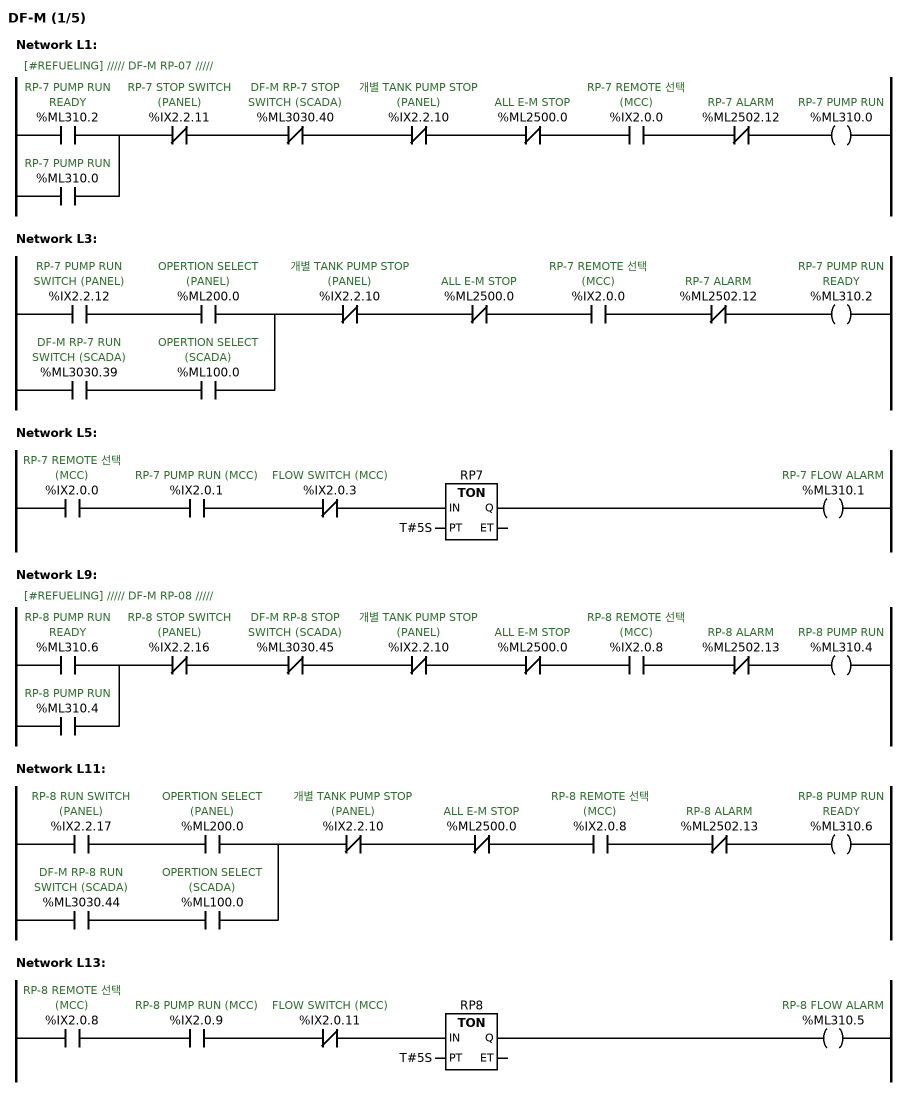
(* [#REFUELING] ///// DF-M RP-07 ///// *)
(* Rung L1 *)
%ML310.0 := (%ML310.2 OR %ML310.0) AND NOT %IX2.2.11 AND NOT %ML3030.40 AND NOT %IX2.2.10 AND NOT %ML2500.0 AND %IX2.0.0 AND NOT %ML2502.12;
(* Rung L3 *)
%ML310.2 := ((%IX2.2.12 AND %ML200.0) OR (%ML3030.39 AND %ML100.0)) AND NOT %IX2.2.10 AND NOT %ML2500.0 AND %IX2.0.0 AND NOT %ML2502.12;
(* Rung L5 *)
RP7(IN := %IX2.0.0 AND %IX2.0.1 AND NOT %IX2.0.3, PT := T#5S);
%ML310.1 := RP7.Q;
(* [#REFUELING] ///// DF-M RP-08 ///// *)
(* Rung L9 *)
%ML310.4 := (%ML310.6 OR %ML310.4) AND NOT %IX2.2.16 AND NOT %ML3030.45 AND NOT %IX2.2.10 AND NOT %ML2500.0 AND %IX2.0.8 AND NOT %ML2502.13;
(* Rung L11 *)
%ML310.6 := ((%IX2.2.17 AND %ML200.0) OR (%ML3030.44 AND %ML100.0)) AND NOT %IX2.2.10 AND NOT %ML2500.0 AND %IX2.0.8 AND NOT %ML2502.13;
(* Rung L13 *)
RP8(IN := %IX2.0.8 AND %IX2.0.9 AND NOT %IX2.0.11, PT := T#5S);
%ML310.5 := RP8.Q;

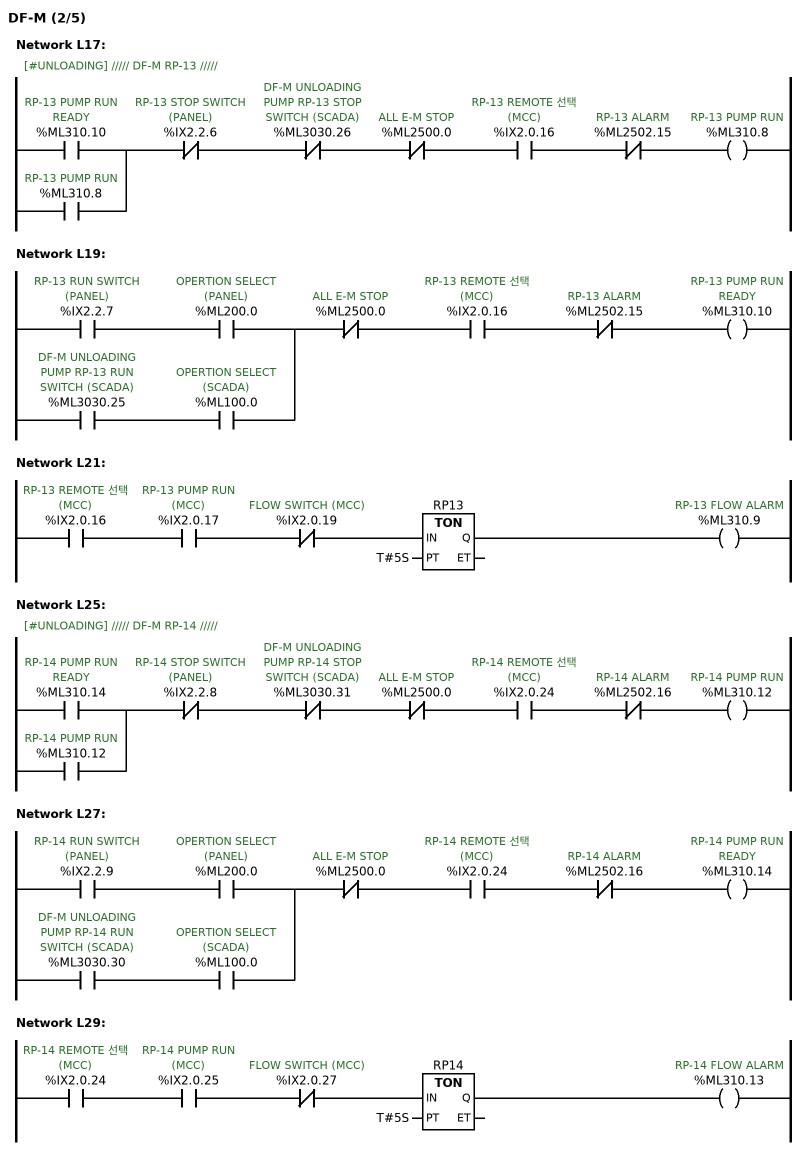
(* [#UNLOADING] ///// DF-M RP-13 ///// *)
(* Rung L17 *)
%ML310.8 := (%ML310.10 OR %ML310.8) AND NOT %IX2.2.6 AND NOT %ML3030.26 AND NOT %ML2500.0 AND %IX2.0.16 AND NOT %ML2502.15;
(* Rung L19 *)
%ML310.10 := ((%IX2.2.7 AND %ML200.0) OR (%ML3030.25 AND %ML100.0)) AND NOT %ML2500.0 AND %IX2.0.16 AND NOT %ML2502.15;
(* Rung L21 *)
RP13(IN := %IX2.0.16 AND %IX2.0.17 AND NOT %IX2.0.19, PT := T#5S);
%ML310.9 := RP13.Q;
(* [#UNLOADING] ///// DF-M RP-14 ///// *)
(* Rung L25 *)
%ML310.12 := (%ML310.14 OR %ML310.12) AND NOT %IX2.2.8 AND NOT %ML3030.31 AND NOT %ML2500.0 AND %IX2.0.24 AND NOT %ML2502.16;
(* Rung L27 *)
%ML310.14 := ((%IX2.2.9 AND %ML200.0) OR (%ML3030.30 AND %ML100.0)) AND NOT %ML2500.0 AND %IX2.0.24 AND NOT %ML2502.16;
(* Rung L29 *)
RP14(IN := %IX2.0.24 AND %IX2.0.25 AND NOT %IX2.0.27, PT := T#5S);
%ML310.13 := RP14.Q;

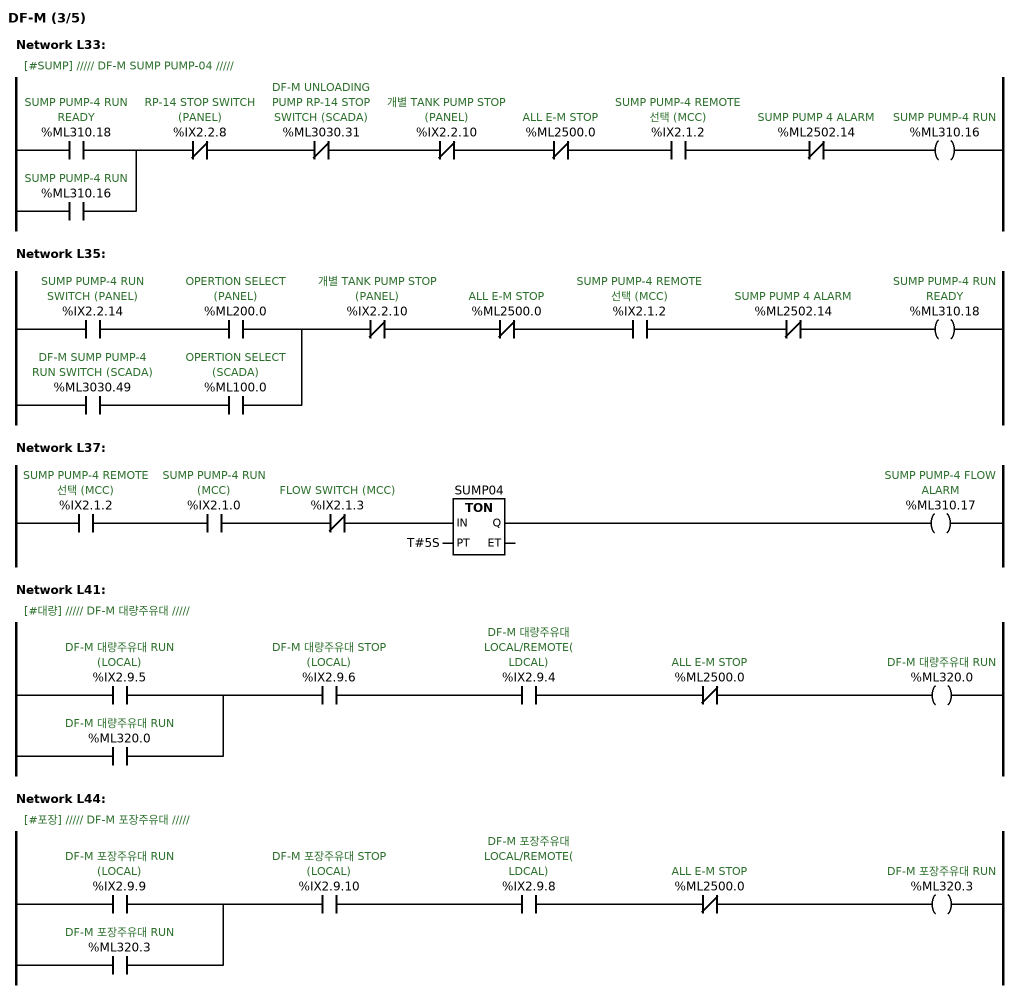
(* [#SUMP] ///// DF-M SUMP PUMP-04 ///// *)
(* Rung L33 *)
%ML310.16 := (%ML310.18 OR %ML310.16) AND NOT %IX2.2.8 AND NOT %ML3030.31 AND NOT %IX2.2.10 AND NOT %ML2500.0 AND %IX2.1.2 AND NOT %ML2502.14;
(* Rung L35 *)
%ML310.18 := ((%IX2.2.14 AND %ML200.0) OR (%ML3030.49 AND %ML100.0)) AND NOT %IX2.2.10 AND NOT %ML2500.0 AND %IX2.1.2 AND NOT %ML2502.14;
(* Rung L37 *)
SUMP04(IN := %IX2.1.2 AND %IX2.1.0 AND NOT %IX2.1.3, PT := T#5S);
%ML310.17 := SUMP04.Q;
(* [#대량] ///// DF-M 대량주유대 ///// *)
(* Rung L41 *)
%ML320.0 := (%IX2.9.5 OR %ML320.0) AND %IX2.9.6 AND %IX2.9.4 AND NOT %ML2500.0;
(* [#포장] ///// DF-M 포장주유대 ///// *)
(* Rung L44 *)
%ML320.3 := (%IX2.9.9 OR %ML320.3) AND %IX2.9.10 AND %IX2.9.8 AND NOT %ML2500.0;

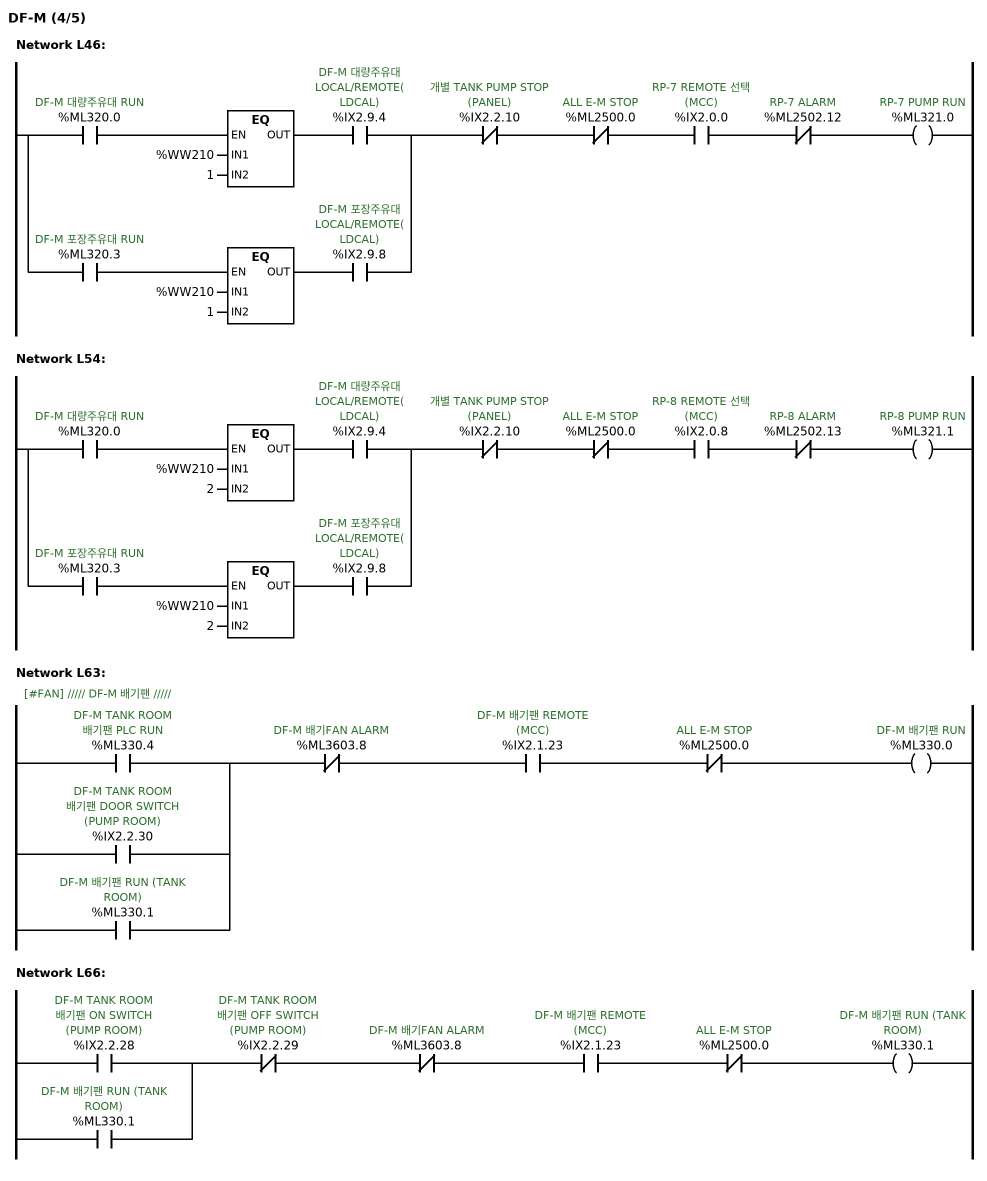
(* Rung L46 *)
IF %ML320.0 THEN _t1 := %WW210 = 1; END_IF;
IF %ML320.3 THEN _t2 := %WW210 = 1; END_IF;
%ML321.0 := ((_t1 AND %IX2.9.4) OR (_t2 AND %IX2.9.8)) AND NOT %IX2.2.10 AND NOT %ML2500.0 AND %IX2.0.0 AND NOT %ML2502.12;
(* Rung L54 *)
IF %ML320.0 THEN _t3 := %WW210 = 2; END_IF;
IF %ML320.3 THEN _t4 := %WW210 = 2; END_IF;
%ML321.1 := ((_t3 AND %IX2.9.4) OR (_t4 AND %IX2.9.8)) AND NOT %IX2.2.10 AND NOT %ML2500.0 AND %IX2.0.8 AND NOT %ML2502.13;
(* [#FAN] ///// DF-M 배기팬 ///// *)
(* Rung L63 *)
%ML330.0 := (%ML330.4 OR %IX2.2.30 OR %ML330.1) AND NOT %ML3603.8 AND %IX2.1.23 AND NOT %ML2500.0;
(* Rung L66 *)
%ML330.1 := (%IX2.2.28 OR %ML330.1) AND NOT %IX2.2.29 AND NOT %ML3603.8 AND %IX2.1.23 AND NOT %ML2500.0;

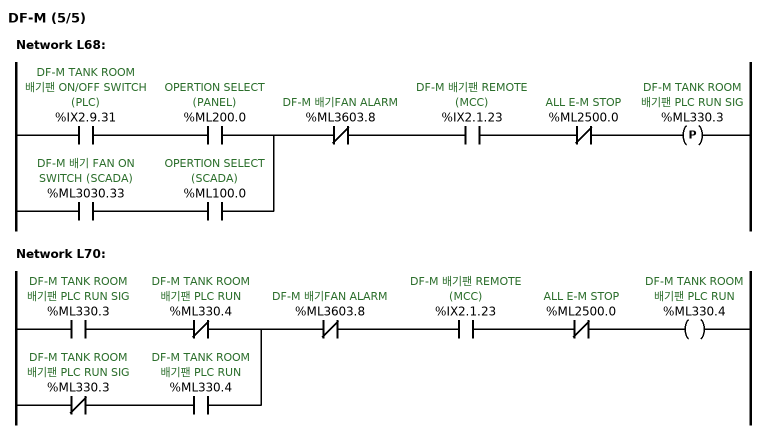
(* Rung L68 *)
_e5(CLK := ((%IX2.9.31 AND %ML200.0) OR (%ML3030.33 AND %ML100.0)) AND NOT %ML3603.8 AND %IX2.1.23 AND NOT %ML2500.0);
%ML330.3 := _e5.Q;
(* Rung L70 *)
%ML330.4 := ((%ML330.3 AND NOT %ML330.4) OR (NOT %ML330.3 AND %ML330.4)) AND NOT %ML3603.8 AND %IX2.1.23 AND NOT %ML2500.0;
END_PROGRAM

PROGRAM MOGAS (* task: 스캔 프로그램 *)
VAR
    DP01 : TON; (* DRAIN PUMP FLOW SENSOR *)
    RP10 : TON;
    RP11 : TON;
    RP12 : TON;
    RP13 : TON;
    RP14 : TON;
    RP15 : TON;
    RP16 : TON;
    RP5 : TON;
    RP6 : TON;
    RP7 : TON;
    RP8 : TON;
    RP9 : TON;
    SUMP04 : TON;
END_VAR
VAR
    _t1 : BOOL;
    _t2 : BOOL;
    _t3 : BOOL;
    _t4 : BOOL;
    _e5 : R_TRIG;
END_VAR

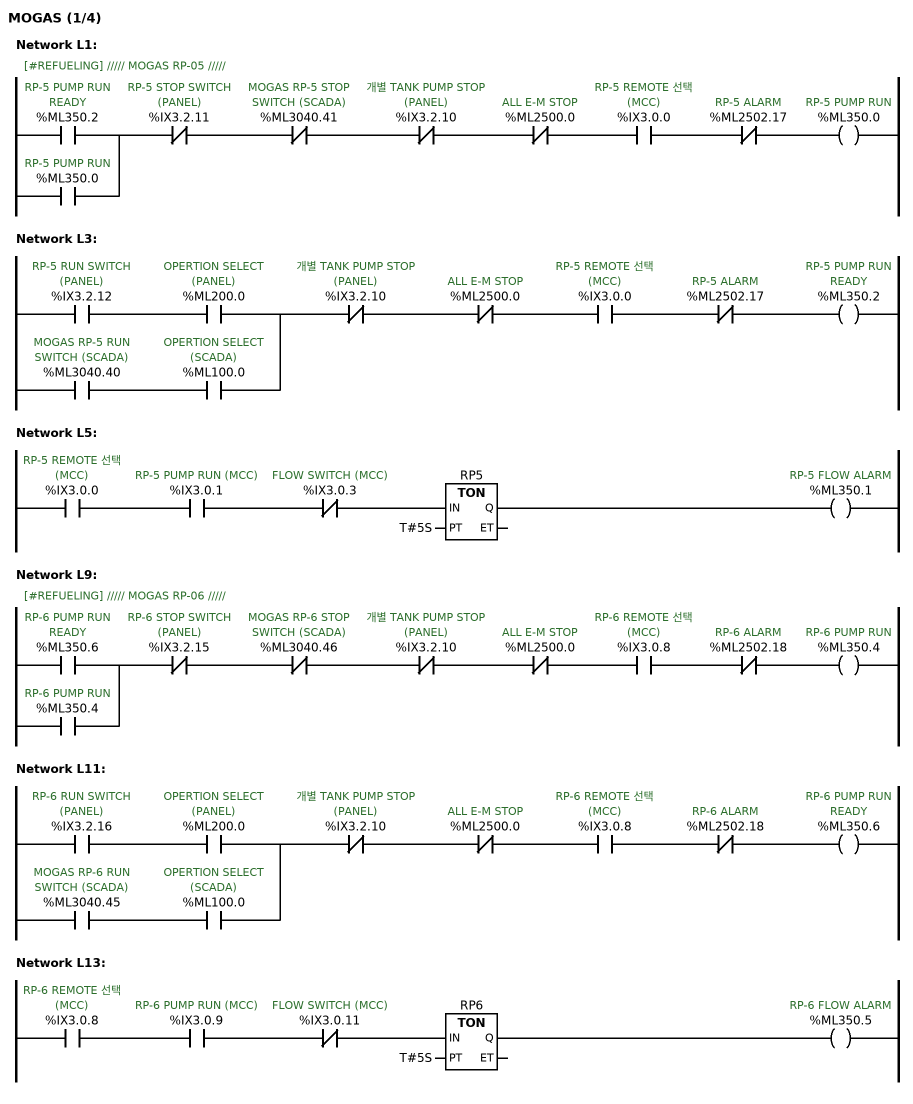
(* [#REFUELING] ///// MOGAS RP-05 ///// *)
(* Rung L1 *)
%ML350.0 := (%ML350.2 OR %ML350.0) AND NOT %IX3.2.11 AND NOT %ML3040.41 AND NOT %IX3.2.10 AND NOT %ML2500.0 AND %IX3.0.0 AND NOT %ML2502.17;
(* Rung L3 *)
%ML350.2 := ((%IX3.2.12 AND %ML200.0) OR (%ML3040.40 AND %ML100.0)) AND NOT %IX3.2.10 AND NOT %ML2500.0 AND %IX3.0.0 AND NOT %ML2502.17;
(* Rung L5 *)
RP5(IN := %IX3.0.0 AND %IX3.0.1 AND NOT %IX3.0.3, PT := T#5S);
%ML350.1 := RP5.Q;
(* [#REFUELING] ///// MOGAS RP-06 ///// *)
(* Rung L9 *)
%ML350.4 := (%ML350.6 OR %ML350.4) AND NOT %IX3.2.15 AND NOT %ML3040.46 AND NOT %IX3.2.10 AND NOT %ML2500.0 AND %IX3.0.8 AND NOT %ML2502.18;
(* Rung L11 *)
%ML350.6 := ((%IX3.2.16 AND %ML200.0) OR (%ML3040.45 AND %ML100.0)) AND NOT %IX3.2.10 AND NOT %ML2500.0 AND %IX3.0.8 AND NOT %ML2502.18;
(* Rung L13 *)
RP6(IN := %IX3.0.8 AND %IX3.0.9 AND NOT %IX3.0.11, PT := T#5S);
%ML350.5 := RP6.Q;

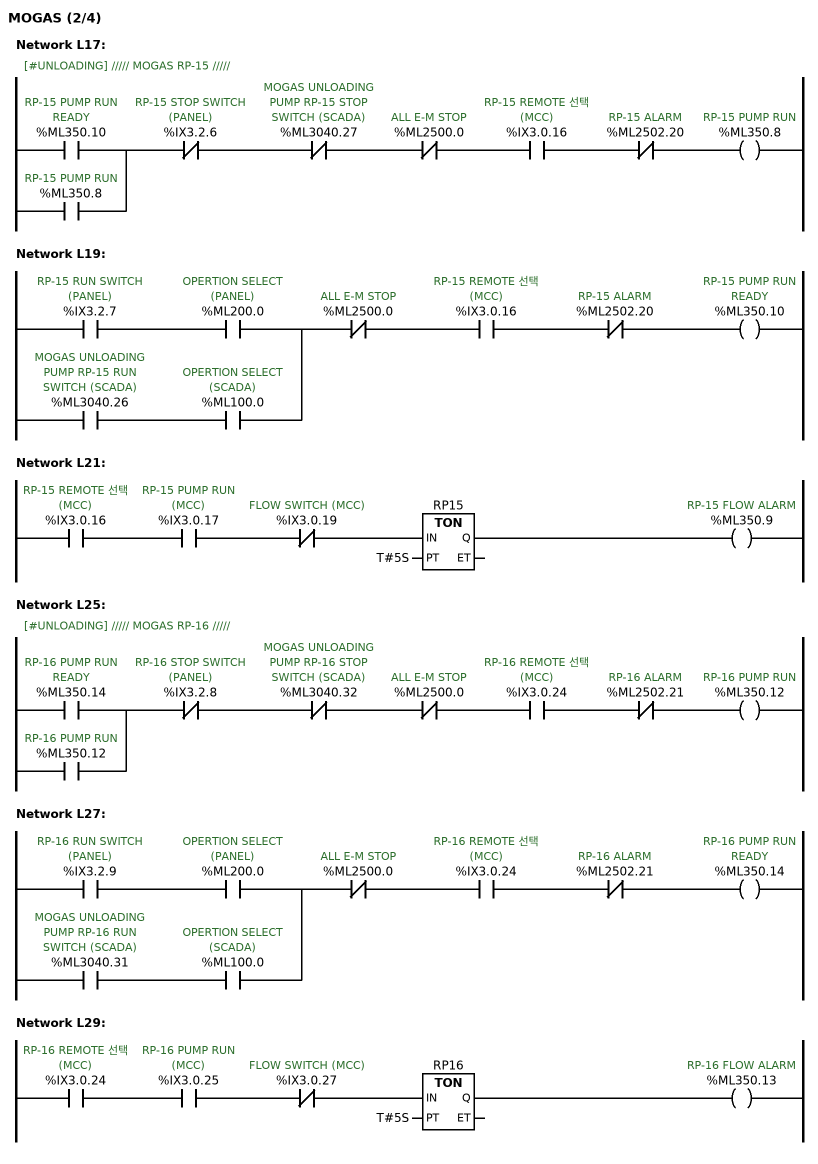
(* [#UNLOADING] ///// MOGAS RP-15 ///// *)
(* Rung L17 *)
%ML350.8 := (%ML350.10 OR %ML350.8) AND NOT %IX3.2.6 AND NOT %ML3040.27 AND NOT %ML2500.0 AND %IX3.0.16 AND NOT %ML2502.20;
(* Rung L19 *)
%ML350.10 := ((%IX3.2.7 AND %ML200.0) OR (%ML3040.26 AND %ML100.0)) AND NOT %ML2500.0 AND %IX3.0.16 AND NOT %ML2502.20;
(* Rung L21 *)
RP15(IN := %IX3.0.16 AND %IX3.0.17 AND NOT %IX3.0.19, PT := T#5S);
%ML350.9 := RP15.Q;
(* [#UNLOADING] ///// MOGAS RP-16 ///// *)
(* Rung L25 *)
%ML350.12 := (%ML350.14 OR %ML350.12) AND NOT %IX3.2.8 AND NOT %ML3040.32 AND NOT %ML2500.0 AND %IX3.0.24 AND NOT %ML2502.21;
(* Rung L27 *)
%ML350.14 := ((%IX3.2.9 AND %ML200.0) OR (%ML3040.31 AND %ML100.0)) AND NOT %ML2500.0 AND %IX3.0.24 AND NOT %ML2502.21;
(* Rung L29 *)
RP16(IN := %IX3.0.24 AND %IX3.0.25 AND NOT %IX3.0.27, PT := T#5S);
%ML350.13 := RP16.Q;

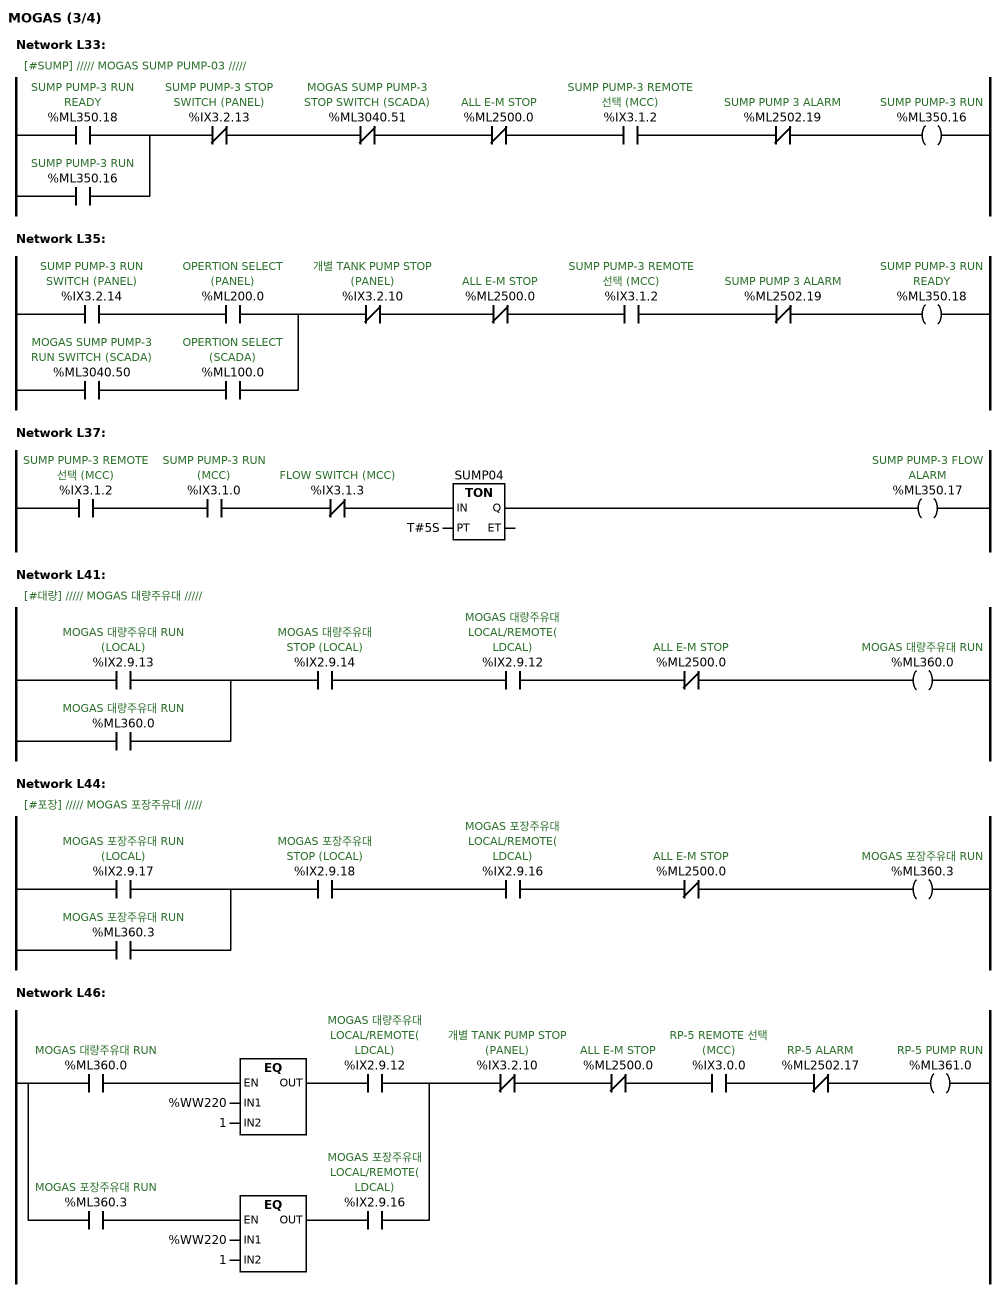
(* [#SUMP] ///// MOGAS SUMP PUMP-03 ///// *)
(* Rung L33 *)
%ML350.16 := (%ML350.18 OR %ML350.16) AND NOT %IX3.2.13 AND NOT %ML3040.51 AND NOT %ML2500.0 AND %IX3.1.2 AND NOT %ML2502.19;
(* Rung L35 *)
%ML350.18 := ((%IX3.2.14 AND %ML200.0) OR (%ML3040.50 AND %ML100.0)) AND NOT %IX3.2.10 AND NOT %ML2500.0 AND %IX3.1.2 AND NOT %ML2502.19;
(* Rung L37 *)
SUMP04(IN := %IX3.1.2 AND %IX3.1.0 AND NOT %IX3.1.3, PT := T#5S);
%ML350.17 := SUMP04.Q;
(* [#대량] ///// MOGAS 대량주유대 ///// *)
(* Rung L41 *)
%ML360.0 := (%IX2.9.13 OR %ML360.0) AND %IX2.9.14 AND %IX2.9.12 AND NOT %ML2500.0;
(* [#포장] ///// MOGAS 포장주유대 ///// *)
(* Rung L44 *)
%ML360.3 := (%IX2.9.17 OR %ML360.3) AND %IX2.9.18 AND %IX2.9.16 AND NOT %ML2500.0;
(* Rung L46 *)
IF %ML360.0 THEN _t1 := %WW220 = 1; END_IF;
IF %ML360.3 THEN _t2 := %WW220 = 1; END_IF;
%ML361.0 := ((_t1 AND %IX2.9.12) OR (_t2 AND %IX2.9.16)) AND NOT %IX3.2.10 AND NOT %ML2500.0 AND %IX3.0.0 AND NOT %ML2502.17;

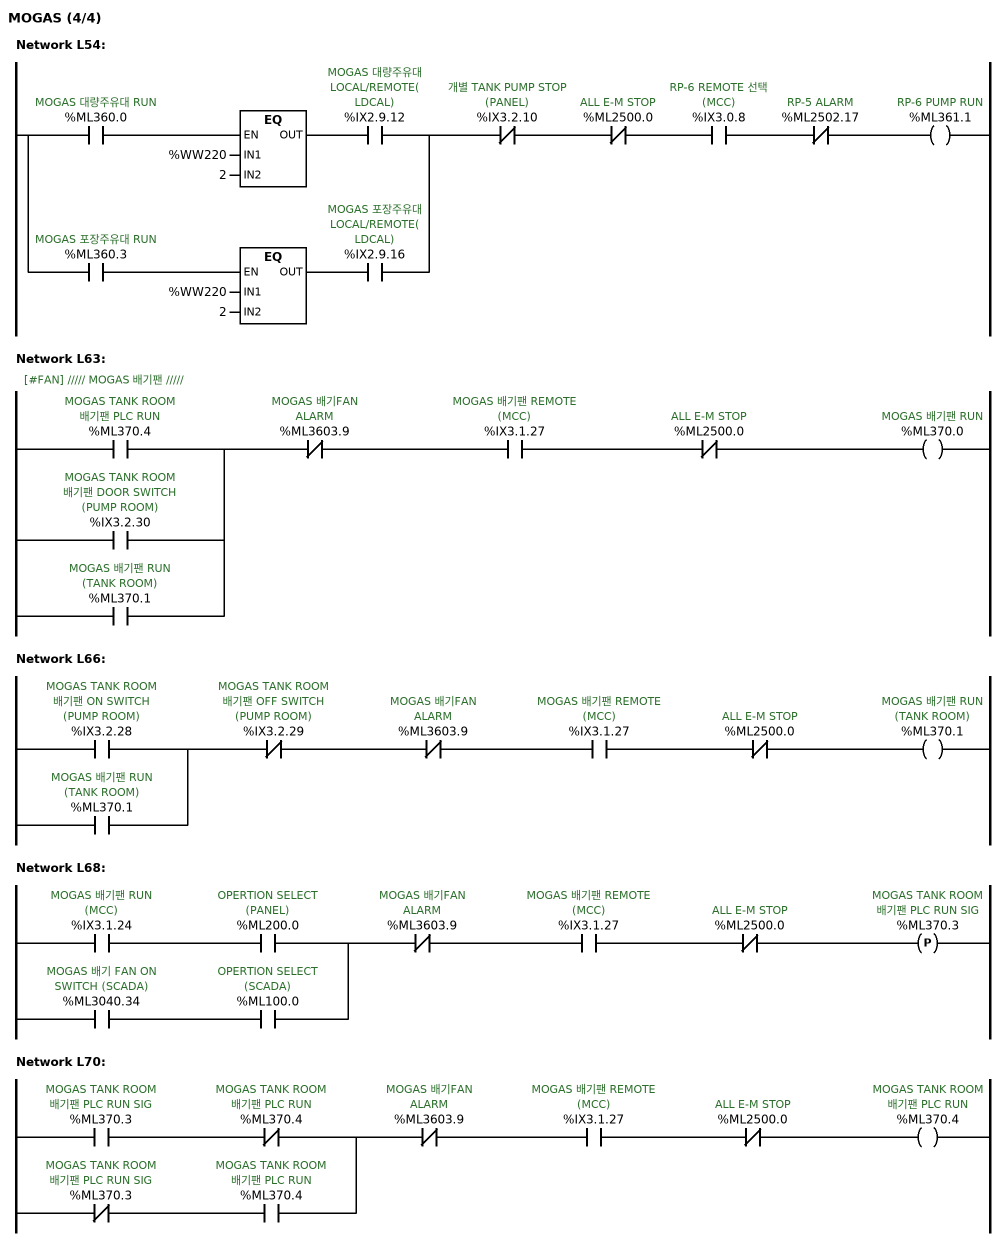
(* Rung L54 *)
IF %ML360.0 THEN _t3 := %WW220 = 2; END_IF;
IF %ML360.3 THEN _t4 := %WW220 = 2; END_IF;
%ML361.1 := ((_t3 AND %IX2.9.12) OR (_t4 AND %IX2.9.16)) AND NOT %IX3.2.10 AND NOT %ML2500.0 AND %IX3.0.8 AND NOT %ML2502.17;
(* [#FAN] ///// MOGAS 배기팬 ///// *)
(* Rung L63 *)
%ML370.0 := (%ML370.4 OR %IX3.2.30 OR %ML370.1) AND NOT %ML3603.9 AND %IX3.1.27 AND NOT %ML2500.0;
(* Rung L66 *)
%ML370.1 := (%IX3.2.28 OR %ML370.1) AND NOT %IX3.2.29 AND NOT %ML3603.9 AND %IX3.1.27 AND NOT %ML2500.0;
(* Rung L68 *)
_e5(CLK := ((%IX3.1.24 AND %ML200.0) OR (%ML3040.34 AND %ML100.0)) AND NOT %ML3603.9 AND %IX3.1.27 AND NOT %ML2500.0);
%ML370.3 := _e5.Q;
(* Rung L70 *)
%ML370.4 := ((%ML370.3 AND NOT %ML370.4) OR (NOT %ML370.3 AND %ML370.4)) AND NOT %ML3603.9 AND %IX3.1.27 AND NOT %ML2500.0;
END_PROGRAM

PROGRAM ANALOGUE (* task: 스캔 프로그램 *)
VAR
    DF1A_LEVEL_PER : INT;
    DF1B_LEVEL_PER : INT;
    DFM_LEVEL_PER : INT;
    DTK1_LEVEL_PER : INT;
    DTK2_LEVEL_PER : INT;
    FIT_1 : INT;
    FIT_2 : INT;
    MOGAS_LEVEL_PER : INT;
END_VAR
VAR_EXTERNAL
    _0108_CH0_ACT : BOOL; (* AT %UX1.8.16 *) (* 절연형 아날로그입력 모듈: 채널0 운전중 *)
    _0108_CH0_DATA : INT; (* AT %UW1.8.2 *) (* 절연형 아날로그입력 모듈: 채널0 변환값 *)
    _0108_CH0_IDD : BOOL; (* AT %UX1.8.160 *) (* 절연형 아날로그입력 모듈: 채널0 입력단선검출 *)
    _0108_CH1_ACT : BOOL; (* AT %UX1.8.17 *) (* 절연형 아날로그입력 모듈: 채널1 운전중 *)
    _0108_CH1_DATA : INT; (* AT %UW1.8.3 *) (* 절연형 아날로그입력 모듈: 채널1 변환값 *)
    _0108_CH1_IDD : BOOL; (* AT %UX1.8.161 *) (* 절연형 아날로그입력 모듈: 채널1 입력단선검출 *)
    _0108_CH2_ACT : BOOL; (* AT %UX1.8.18 *) (* 절연형 아날로그입력 모듈: 채널2 운전중 *)
    _0108_CH2_DATA : INT; (* AT %UW1.8.4 *) (* 절연형 아날로그입력 모듈: 채널2 변환값 *)
    _0108_CH2_IDD : BOOL; (* AT %UX1.8.162 *) (* 절연형 아날로그입력 모듈: 채널2 입력단선검출 *)
    _0108_CH3_ACT : BOOL; (* AT %UX1.8.19 *) (* 절연형 아날로그입력 모듈: 채널3 운전중 *)
    _0108_CH3_DATA : INT; (* AT %UW1.8.5 *) (* 절연형 아날로그입력 모듈: 채널3 변환값 *)
    _0108_CH3_IDD : BOOL; (* AT %UX1.8.163 *) (* 절연형 아날로그입력 모듈: 채널3 입력단선검출 *)
    _0109_CH0_ACT : BOOL; (* AT %UX1.9.16 *) (* 절연형 아날로그출력 모듈: 채널0 운전중 *)
    _0109_CH0_DATA : INT; (* AT %UW1.9.3 *) (* 절연형 아날로그출력 모듈: 채널0 입력값 *)
    _0109_CH0_ERR : BOOL; (* AT %UX1.9.0 *) (* 절연형 아날로그출력 모듈: 채널0 에러 *)
    _0109_CH0_OUTEN : BOOL; (* AT %UX1.9.32 *) (* 절연형 아날로그출력 모듈: 채널0 출력상태설정 *)
    _0109_CH1_ACT : BOOL; (* AT %UX1.9.17 *) (* 절연형 아날로그출력 모듈: 채널1 운전중 *)
    _0109_CH1_DATA : INT; (* AT %UW1.9.4 *) (* 절연형 아날로그출력 모듈: 채널1 입력값 *)
    _0109_CH1_ERR : BOOL; (* AT %UX1.9.1 *) (* 절연형 아날로그출력 모듈: 채널1 에러 *)
    _0109_CH2_ACT : BOOL; (* AT %UX1.9.18 *) (* 절연형 아날로그출력 모듈: 채널2 운전중 *)
    _0109_CH2_DATA : INT; (* AT %UW1.9.5 *) (* 절연형 아날로그출력 모듈: 채널2 입력값 *)
    _0109_CH3_ACT : BOOL; (* AT %UX1.9.19 *) (* 절연형 아날로그출력 모듈: 채널3 운전중 *)
    _0109_CH3_DATA : INT; (* AT %UW1.9.6 *) (* 절연형 아날로그출력 모듈: 채널3 입력값 *)
    _0109_OUTEN : WORD; (* AT %UW1.9.2 *) (* 절연형 아날로그출력 모듈: 출력상태 설정 *)
    _0110_CH0_ACT : BOOL; (* AT %UX1.10.16 *) (* 절연형 아날로그출력 모듈: 채널0 운전중 *)
    _0110_CH0_DATA : INT; (* AT %UW1.10.3 *) (* 절연형 아날로그출력 모듈: 채널0 입력값 *)
    _0110_CH0_ERR : BOOL; (* AT %UX1.10.0 *) (* 절연형 아날로그출력 모듈: 채널0 에러 *)
    _0110_OUTEN : WORD; (* AT %UW1.10.2 *) (* 절연형 아날로그출력 모듈: 출력상태 설정 *)
    _0206_CH0_ACT : BOOL; (* AT %UX2.6.16 *) (* 절연형 아날로그입력 모듈: 채널0 운전중 *)
    _0206_CH0_DATA : INT; (* AT %UW2.6.2 *) (* 절연형 아날로그입력 모듈: 채널0 변환값 *)
    _0206_CH0_IDD : BOOL; (* AT %UX2.6.160 *) (* 절연형 아날로그입력 모듈: 채널0 입력단선검출 *)
    _0206_CH1_ACT : BOOL; (* AT %UX2.6.17 *) (* 절연형 아날로그입력 모듈: 채널1 운전중 *)
    _0206_CH1_DATA : INT; (* AT %UW2.6.3 *) (* 절연형 아날로그입력 모듈: 채널1 변환값 *)
    _0206_CH1_IDD : BOOL; (* AT %UX2.6.161 *) (* 절연형 아날로그입력 모듈: 채널1 입력단선검출 *)
    _0206_CH2_ACT : BOOL; (* AT %UX2.6.18 *) (* 절연형 아날로그입력 모듈: 채널2 운전중 *)
    _0206_CH2_DATA : INT; (* AT %UW2.6.4 *) (* 절연형 아날로그입력 모듈: 채널2 변환값 *)
    _0206_CH2_IDD : BOOL; (* AT %UX2.6.162 *) (* 절연형 아날로그입력 모듈: 채널2 입력단선검출 *)
    _0206_CH3_ACT : BOOL; (* AT %UX2.6.19 *) (* 절연형 아날로그입력 모듈: 채널3 운전중 *)
    _0206_CH3_DATA : INT; (* AT %UW2.6.5 *) (* 절연형 아날로그입력 모듈: 채널3 변환값 *)
    _0206_CH3_IDD : BOOL; (* AT %UX2.6.163 *) (* 절연형 아날로그입력 모듈: 채널3 입력단선검출 *)
    _0207_CH0_ACT : BOOL; (* AT %UX2.7.16 *) (* 절연형 아날로그출력 모듈: 채널0 운전중 *)
    _0207_CH0_DATA : INT; (* AT %UW2.7.3 *) (* 절연형 아날로그출력 모듈: 채널0 입력값 *)
    _0207_CH0_ERR : BOOL; (* AT %UX2.7.0 *) (* 절연형 아날로그출력 모듈: 채널0 에러 *)
    _0207_CH1_ACT : BOOL; (* AT %UX2.7.17 *) (* 절연형 아날로그출력 모듈: 채널1 운전중 *)
    _0207_CH1_DATA : INT; (* AT %UW2.7.4 *) (* 절연형 아날로그출력 모듈: 채널1 입력값 *)
    _0207_CH2_ACT : BOOL; (* AT %UX2.7.18 *) (* 절연형 아날로그출력 모듈: 채널2 운전중 *)
    _0207_CH2_DATA : INT; (* AT %UW2.7.5 *) (* 절연형 아날로그출력 모듈: 채널2 입력값 *)
    _0207_CH3_DATA : INT; (* AT %UW2.7.6 *) (* 절연형 아날로그출력 모듈: 채널3 입력값 *)
    _0207_OUTEN : WORD; (* AT %UW2.7.2 *) (* 절연형 아날로그출력 모듈: 출력상태 설정 *)
    _0307_CH0_ACT : BOOL; (* AT %UX3.7.16 *) (* 절연형 아날로그입력 모듈: 채널0 운전중 *)
    _0307_CH0_DATA : INT; (* AT %UW3.7.2 *) (* 절연형 아날로그입력 모듈: 채널0 변환값 *)
    _0307_CH0_IDD : BOOL; (* AT %UX3.7.160 *) (* 절연형 아날로그입력 모듈: 채널0 입력단선검출 *)
    _0307_CH1_ACT : BOOL; (* AT %UX3.7.17 *) (* 절연형 아날로그입력 모듈: 채널1 운전중 *)
    _0307_CH1_DATA : INT; (* AT %UW3.7.3 *) (* 절연형 아날로그입력 모듈: 채널1 변환값 *)
    _0307_CH1_IDD : BOOL; (* AT %UX3.7.161 *) (* 절연형 아날로그입력 모듈: 채널1 입력단선검출 *)
    _0307_CH2_ACT : BOOL; (* AT %UX3.7.18 *) (* 절연형 아날로그입력 모듈: 채널2 운전중 *)
    _0307_CH2_DATA : INT; (* AT %UW3.7.4 *) (* 절연형 아날로그입력 모듈: 채널2 변환값 *)
    _0307_CH2_IDD : BOOL; (* AT %UX3.7.162 *) (* 절연형 아날로그입력 모듈: 채널2 입력단선검출 *)
    _0307_CH3_DATA : INT; (* AT %UW3.7.5 *) (* 절연형 아날로그입력 모듈: 채널3 변환값 *)
    _0307_CH3_IDD : BOOL; (* AT %UX3.7.163 *) (* 절연형 아날로그입력 모듈: 채널3 입력단선검출 *)
    _0308_CH0_ACT : BOOL; (* AT %UX3.8.16 *) (* 절연형 아날로그출력 모듈: 채널0 운전중 *)
    _0308_CH0_DATA : INT; (* AT %UW3.8.3 *) (* 절연형 아날로그출력 모듈: 채널0 입력값 *)
    _0308_CH1_ACT : BOOL; (* AT %UX3.8.17 *) (* 절연형 아날로그출력 모듈: 채널1 운전중 *)
    _0308_CH1_DATA : INT; (* AT %UW3.8.4 *) (* 절연형 아날로그출력 모듈: 채널1 입력값 *)
    _0308_CH2_ACT : BOOL; (* AT %UX3.8.18 *) (* 절연형 아날로그출력 모듈: 채널2 운전중 *)
    _0308_CH2_DATA : INT; (* AT %UW3.8.5 *) (* 절연형 아날로그출력 모듈: 채널2 입력값 *)
    _0308_CH3_ACT : BOOL; (* AT %UX3.8.19 *) (* 절연형 아날로그출력 모듈: 채널3 운전중 *)
    _0308_CH3_DATA : INT; (* AT %UW3.8.6 *) (* 절연형 아날로그출력 모듈: 채널3 입력값 *)
    _0308_OUTEN : WORD; (* AT %UW3.8.2 *) (* 절연형 아날로그출력 모듈: 출력상태 설정 *)
END_VAR
VAR_EXTERNAL CONSTANT
    _F0308_CH0_DEC_RATE : UINT; (* 절연형 아날로그출력 모듈: 채널0 변화율 감소값 *)
    _F0308_CH0_STAT : UINT; (* 절연형 아날로그출력 모듈: 채널0 이상 상태 출력 설정값 *)
    _F0308_LIMIT_EN : UINT; (* 절연형 아날로그출력 모듈: 출력제한 채널 설정 *)
END_VAR
VAR
    _t1 : BOOL;
    _t2 : BOOL;
    _t3 : BOOL;
    _t4 : BOOL;
    _t5 : BOOL;
    _t6 : BOOL;
    _t7 : BOOL;
    _t8 : BOOL;
    _t9 : BOOL;
    _t10 : BOOL;
    _t11 : BOOL;
    _t12 : BOOL;
    _t13 : BOOL;
END_VAR

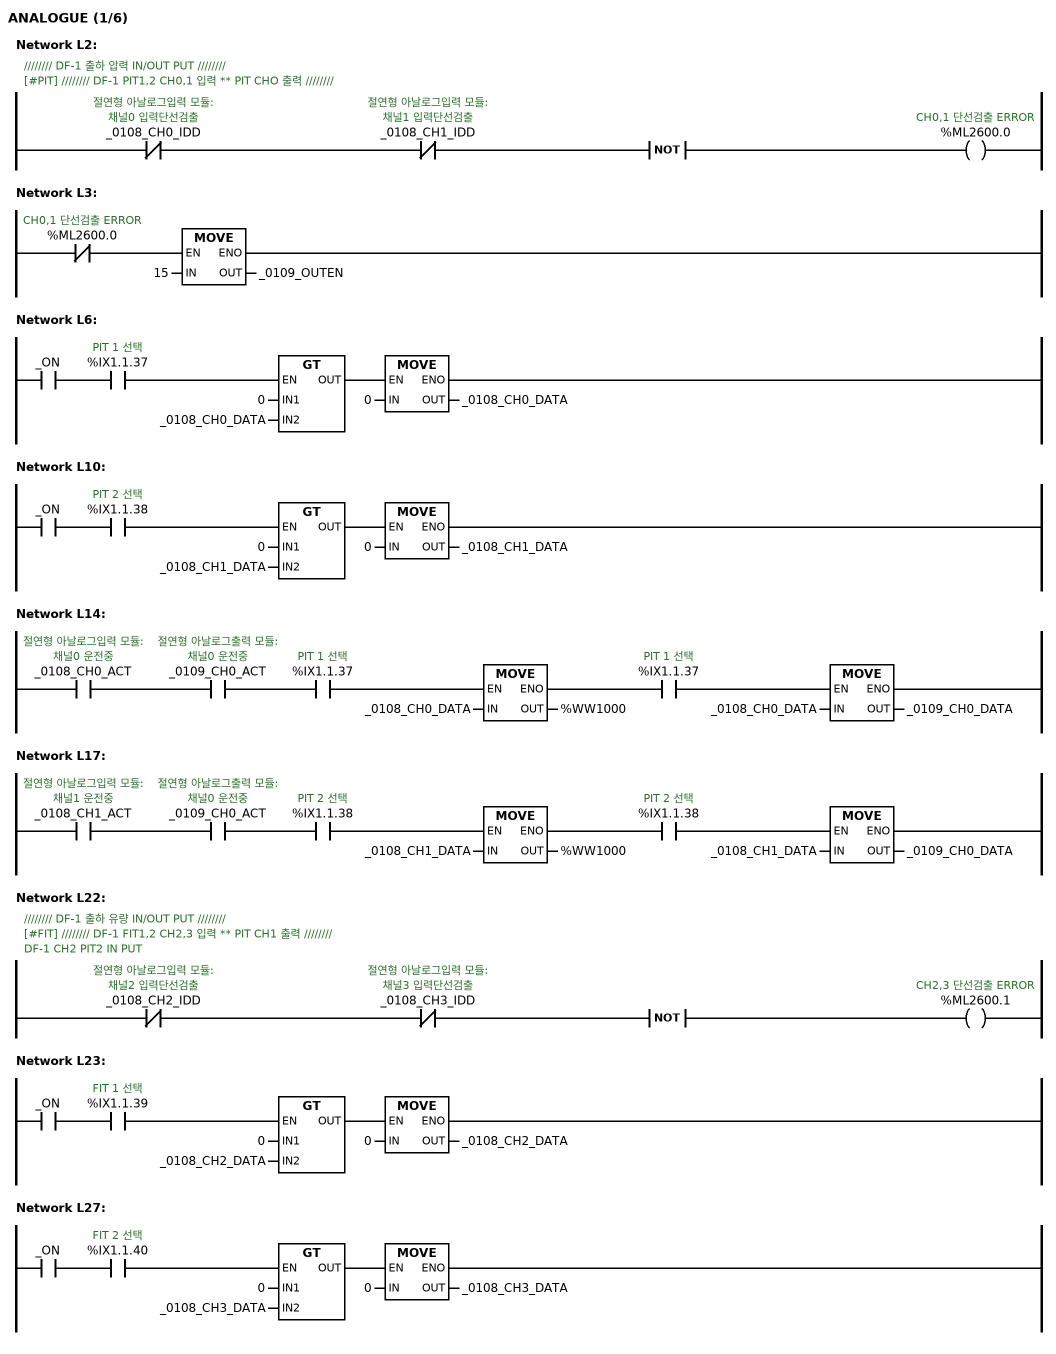
(* //////// DF-1 출하 압력 IN/OUT PUT //////// *)
(* [#PIT] //////// DF-1 PIT1,2 CH0,1 입력 ** PIT CHO 출력 //////// *)
(* Rung L2 *)
%ML2600.0 := NOT (NOT _0108_CH0_IDD AND NOT _0108_CH1_IDD);
(*  *)
(* Rung L3 *)
IF NOT %ML2600.0 THEN _0109_OUTEN := 15; END_IF;
(* Rung L6 *)
IF _ON AND %IX1.1.37 THEN _t1 := 0 > _0108_CH0_DATA; END_IF;
IF _t1 THEN _0108_CH0_DATA := 0; END_IF;
(* Rung L10 *)
IF _ON AND %IX1.1.38 THEN _t2 := 0 > _0108_CH1_DATA; END_IF;
IF _t2 THEN _0108_CH1_DATA := 0; END_IF;
(* Rung L14 *)
IF _0108_CH0_ACT AND _0109_CH0_ACT AND %IX1.1.37 THEN %WW1000 := _0108_CH0_DATA; END_IF;
IF _0108_CH0_ACT AND _0109_CH0_ACT AND %IX1.1.37 AND %IX1.1.37 THEN
    _0109_CH0_DATA := _0108_CH0_DATA;
END_IF;
(* Rung L17 *)
IF _0108_CH1_ACT AND _0109_CH0_ACT AND %IX1.1.38 THEN %WW1000 := _0108_CH1_DATA; END_IF;
IF _0108_CH1_ACT AND _0109_CH0_ACT AND %IX1.1.38 AND %IX1.1.38 THEN
    _0109_CH0_DATA := _0108_CH1_DATA;
END_IF;
(* //////// DF-1 출하 유량 IN/OUT PUT //////// *)
(* [#FIT] //////// DF-1 FIT1,2 CH2,3 입력 ** PIT CH1 출력 //////// *)
(* Rung L22 *)
%ML2600.1 := NOT (NOT _0108_CH2_IDD AND NOT _0108_CH3_IDD);
(* DF-1 CH2 PIT2 IN PUT *)
(* Rung L23 *)
IF _ON AND %IX1.1.39 THEN _t3 := 0 > _0108_CH2_DATA; END_IF;
IF _t3 THEN _0108_CH2_DATA := 0; END_IF;
(* Rung L27 *)
IF _ON AND %IX1.1.40 THEN _t4 := 0 > _0108_CH3_DATA; END_IF;
IF _t4 THEN _0108_CH3_DATA := 0; END_IF;

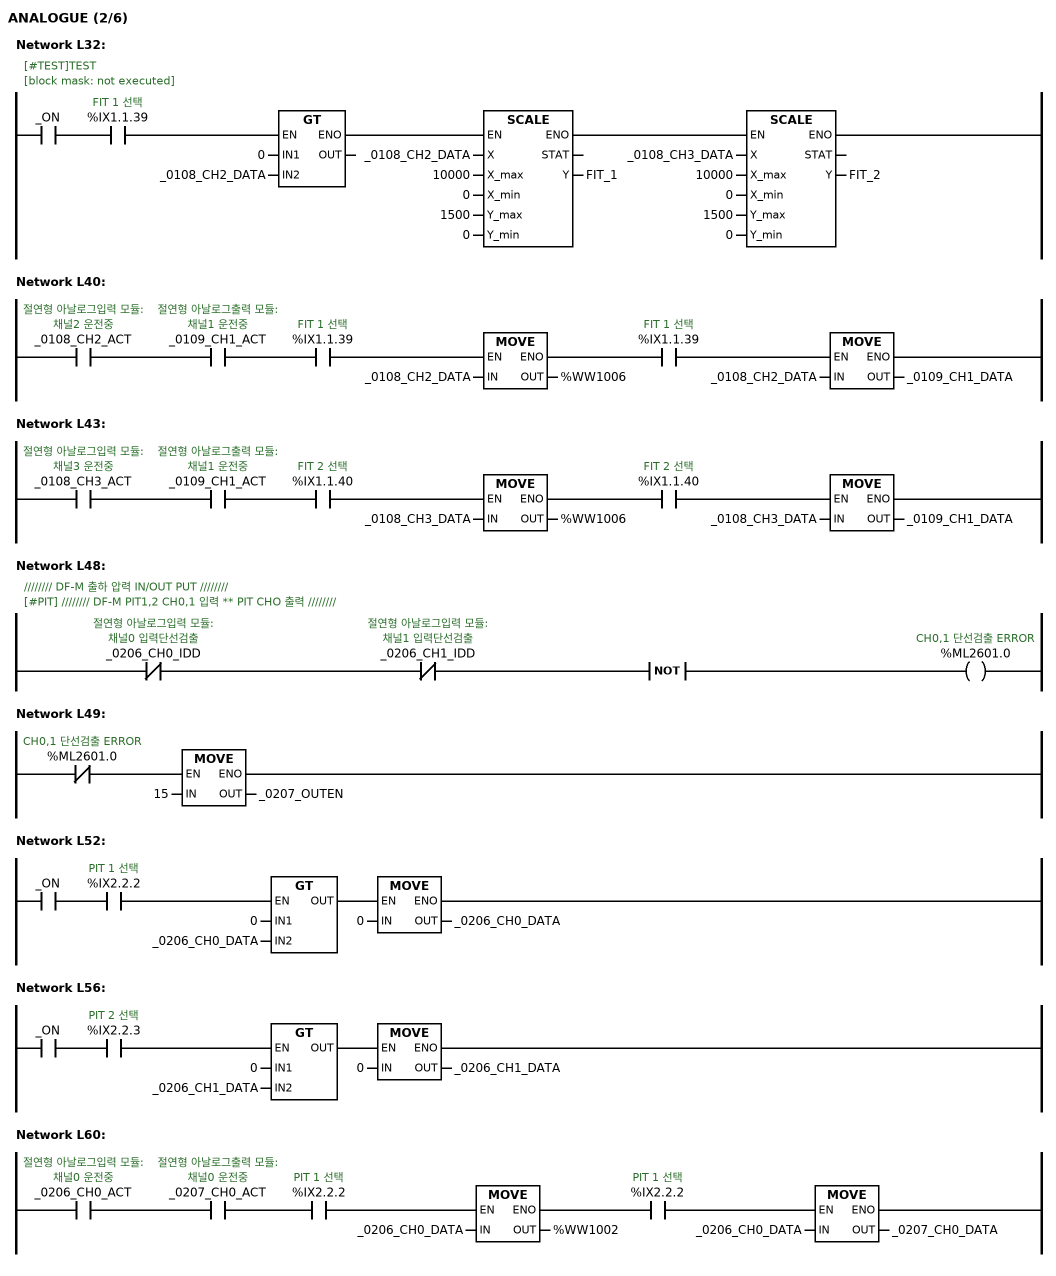
(* [#TEST]TEST *)
(* Rung L32 is block-masked: not executed *)
// IF _ON AND %IX1.1.39 THEN
//     _t5 := 0 > _0108_CH2_DATA;
//     SCALE(X := _0108_CH2_DATA, X_max := 10000, X_min := 0, Y_max := 1500, Y_min := 0, Y => FIT_1);
//     SCALE(X := _0108_CH3_DATA, X_max := 10000, X_min := 0, Y_max := 1500, Y_min := 0, Y => FIT_2);
// END_IF;
(*  *)
(* Rung L40 *)
IF _0108_CH2_ACT AND _0109_CH1_ACT AND %IX1.1.39 THEN %WW1006 := _0108_CH2_DATA; END_IF;
IF _0108_CH2_ACT AND _0109_CH1_ACT AND %IX1.1.39 AND %IX1.1.39 THEN
    _0109_CH1_DATA := _0108_CH2_DATA;
END_IF;
(* Rung L43 *)
IF _0108_CH3_ACT AND _0109_CH1_ACT AND %IX1.1.40 THEN %WW1006 := _0108_CH3_DATA; END_IF;
IF _0108_CH3_ACT AND _0109_CH1_ACT AND %IX1.1.40 AND %IX1.1.40 THEN
    _0109_CH1_DATA := _0108_CH3_DATA;
END_IF;
(* //////// DF-M 출하 압력 IN/OUT PUT //////// *)
(* [#PIT] //////// DF-M PIT1,2 CH0,1 입력 ** PIT CHO 출력 //////// *)
(* Rung L48 *)
%ML2601.0 := NOT (NOT _0206_CH0_IDD AND NOT _0206_CH1_IDD);
(*  *)
(* Rung L49 *)
IF NOT %ML2601.0 THEN _0207_OUTEN := 15; END_IF;
(* Rung L52 *)
IF _ON AND %IX2.2.2 THEN _t6 := 0 > _0206_CH0_DATA; END_IF;
IF _t6 THEN _0206_CH0_DATA := 0; END_IF;
(* Rung L56 *)
IF _ON AND %IX2.2.3 THEN _t7 := 0 > _0206_CH1_DATA; END_IF;
IF _t7 THEN _0206_CH1_DATA := 0; END_IF;
(* Rung L60 *)
IF _0206_CH0_ACT AND _0207_CH0_ACT AND %IX2.2.2 THEN %WW1002 := _0206_CH0_DATA; END_IF;
IF _0206_CH0_ACT AND _0207_CH0_ACT AND %IX2.2.2 AND %IX2.2.2 THEN
    _0207_CH0_DATA := _0206_CH0_DATA;
END_IF;

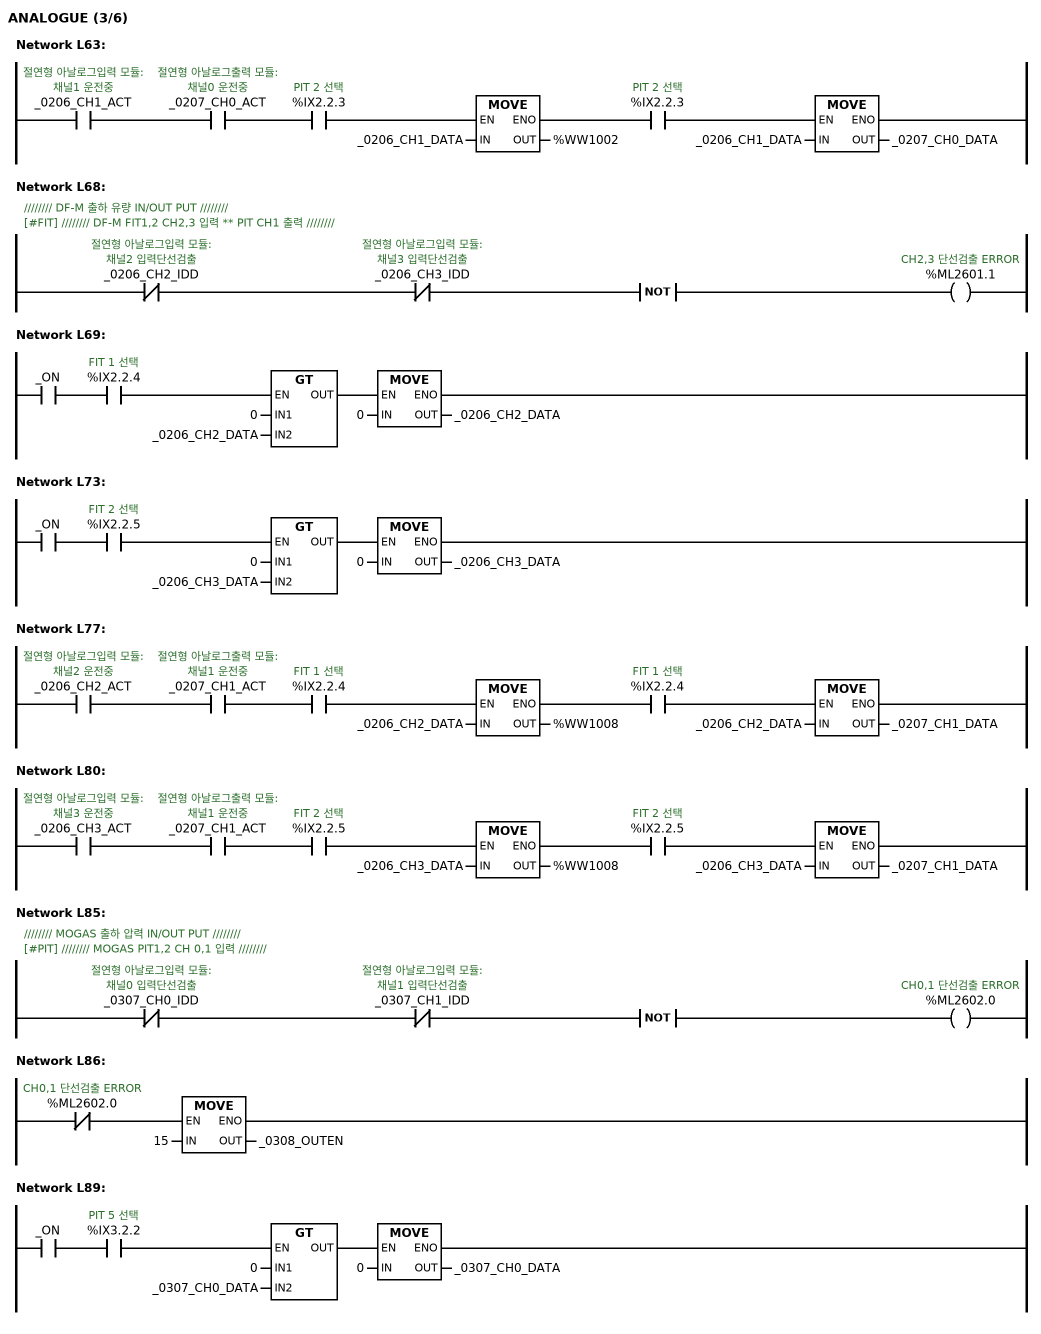
(* Rung L63 *)
IF _0206_CH1_ACT AND _0207_CH0_ACT AND %IX2.2.3 THEN %WW1002 := _0206_CH1_DATA; END_IF;
IF _0206_CH1_ACT AND _0207_CH0_ACT AND %IX2.2.3 AND %IX2.2.3 THEN
    _0207_CH0_DATA := _0206_CH1_DATA;
END_IF;
(* //////// DF-M 출하 유량 IN/OUT PUT //////// *)
(* [#FIT] //////// DF-M FIT1,2 CH2,3 입력 ** PIT CH1 출력 //////// *)
(* Rung L68 *)
%ML2601.1 := NOT (NOT _0206_CH2_IDD AND NOT _0206_CH3_IDD);
(*  *)
(* Rung L69 *)
IF _ON AND %IX2.2.4 THEN _t8 := 0 > _0206_CH2_DATA; END_IF;
IF _t8 THEN _0206_CH2_DATA := 0; END_IF;
(* Rung L73 *)
IF _ON AND %IX2.2.5 THEN _t9 := 0 > _0206_CH3_DATA; END_IF;
IF _t9 THEN _0206_CH3_DATA := 0; END_IF;
(* Rung L77 *)
IF _0206_CH2_ACT AND _0207_CH1_ACT AND %IX2.2.4 THEN %WW1008 := _0206_CH2_DATA; END_IF;
IF _0206_CH2_ACT AND _0207_CH1_ACT AND %IX2.2.4 AND %IX2.2.4 THEN
    _0207_CH1_DATA := _0206_CH2_DATA;
END_IF;
(* Rung L80 *)
IF _0206_CH3_ACT AND _0207_CH1_ACT AND %IX2.2.5 THEN %WW1008 := _0206_CH3_DATA; END_IF;
IF _0206_CH3_ACT AND _0207_CH1_ACT AND %IX2.2.5 AND %IX2.2.5 THEN
    _0207_CH1_DATA := _0206_CH3_DATA;
END_IF;
(* //////// MOGAS 출하 압력 IN/OUT PUT //////// *)
(* [#PIT] //////// MOGAS PIT1,2 CH 0,1 입력 //////// *)
(* Rung L85 *)
%ML2602.0 := NOT (NOT _0307_CH0_IDD AND NOT _0307_CH1_IDD);
(*  *)
(* Rung L86 *)
IF NOT %ML2602.0 THEN _0308_OUTEN := 15; END_IF;
(* Rung L89 *)
IF _ON AND %IX3.2.2 THEN _t10 := 0 > _0307_CH0_DATA; END_IF;
IF _t10 THEN _0307_CH0_DATA := 0; END_IF;

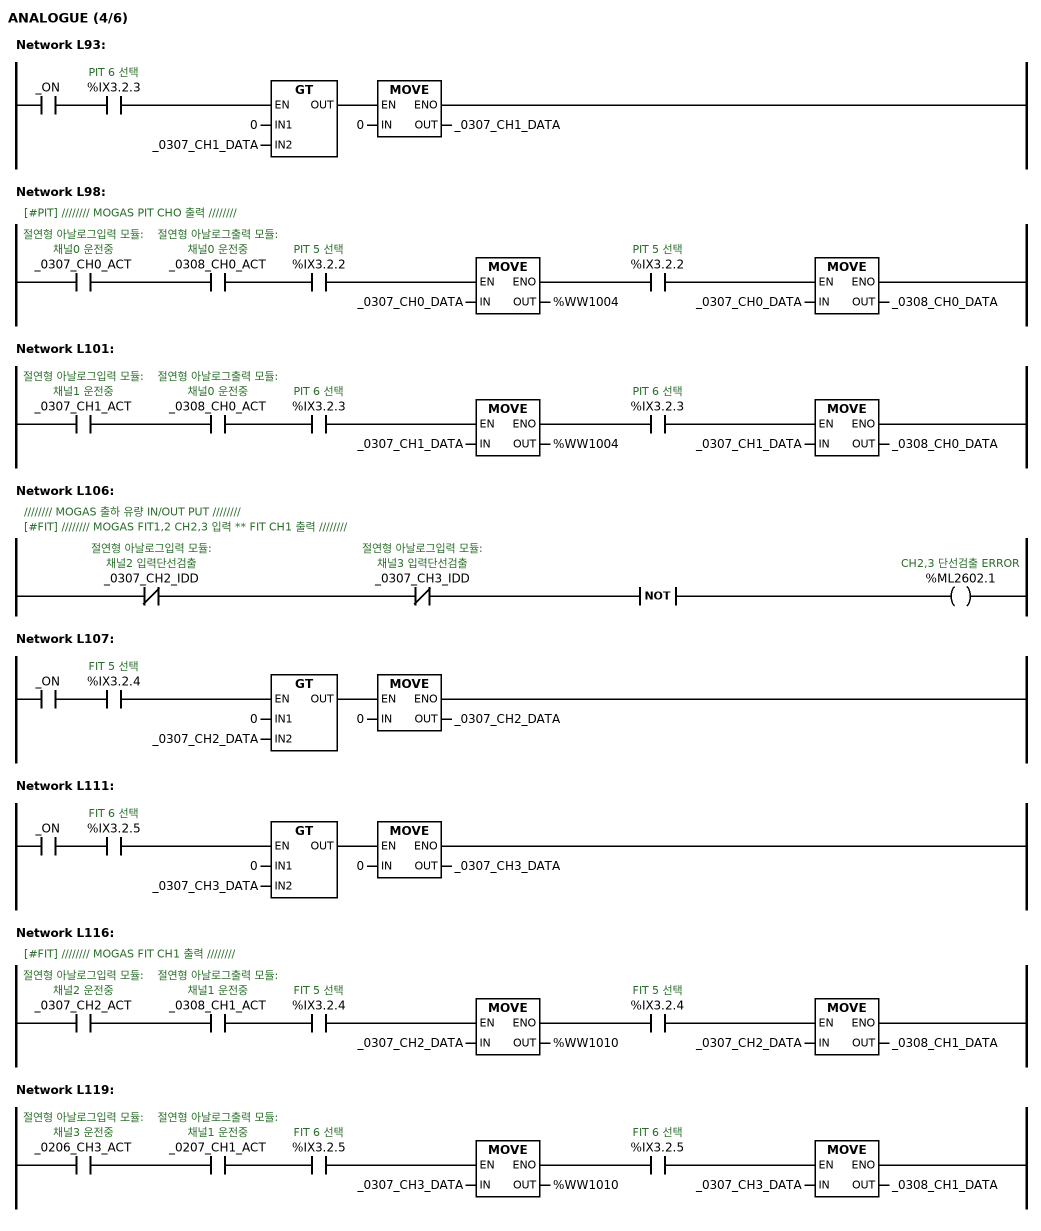
(* Rung L93 *)
IF _ON AND %IX3.2.3 THEN _t11 := 0 > _0307_CH1_DATA; END_IF;
IF _t11 THEN _0307_CH1_DATA := 0; END_IF;
(* [#PIT] //////// MOGAS PIT CHO 출력 //////// *)
(* Rung L98 *)
IF _0307_CH0_ACT AND _0308_CH0_ACT AND %IX3.2.2 THEN %WW1004 := _0307_CH0_DATA; END_IF;
IF _0307_CH0_ACT AND _0308_CH0_ACT AND %IX3.2.2 AND %IX3.2.2 THEN
    _0308_CH0_DATA := _0307_CH0_DATA;
END_IF;
(* Rung L101 *)
IF _0307_CH1_ACT AND _0308_CH0_ACT AND %IX3.2.3 THEN %WW1004 := _0307_CH1_DATA; END_IF;
IF _0307_CH1_ACT AND _0308_CH0_ACT AND %IX3.2.3 AND %IX3.2.3 THEN
    _0308_CH0_DATA := _0307_CH1_DATA;
END_IF;
(* //////// MOGAS 출하 유량 IN/OUT PUT //////// *)
(* [#FIT] //////// MOGAS FIT1,2 CH2,3 입력 ** FIT CH1 출력 //////// *)
(* Rung L106 *)
%ML2602.1 := NOT (NOT _0307_CH2_IDD AND NOT _0307_CH3_IDD);
(*  *)
(* Rung L107 *)
IF _ON AND %IX3.2.4 THEN _t12 := 0 > _0307_CH2_DATA; END_IF;
IF _t12 THEN _0307_CH2_DATA := 0; END_IF;
(* Rung L111 *)
IF _ON AND %IX3.2.5 THEN _t13 := 0 > _0307_CH3_DATA; END_IF;
IF _t13 THEN _0307_CH3_DATA := 0; END_IF;
(* [#FIT] //////// MOGAS FIT CH1 출력 //////// *)
(* Rung L116 *)
IF _0307_CH2_ACT AND _0308_CH1_ACT AND %IX3.2.4 THEN %WW1010 := _0307_CH2_DATA; END_IF;
IF _0307_CH2_ACT AND _0308_CH1_ACT AND %IX3.2.4 AND %IX3.2.4 THEN
    _0308_CH1_DATA := _0307_CH2_DATA;
END_IF;
(* Rung L119 *)
IF _0206_CH3_ACT AND _0207_CH1_ACT AND %IX3.2.5 THEN %WW1010 := _0307_CH3_DATA; END_IF;
IF _0206_CH3_ACT AND _0207_CH1_ACT AND %IX3.2.5 AND %IX3.2.5 THEN
    _0308_CH1_DATA := _0307_CH3_DATA;
END_IF;

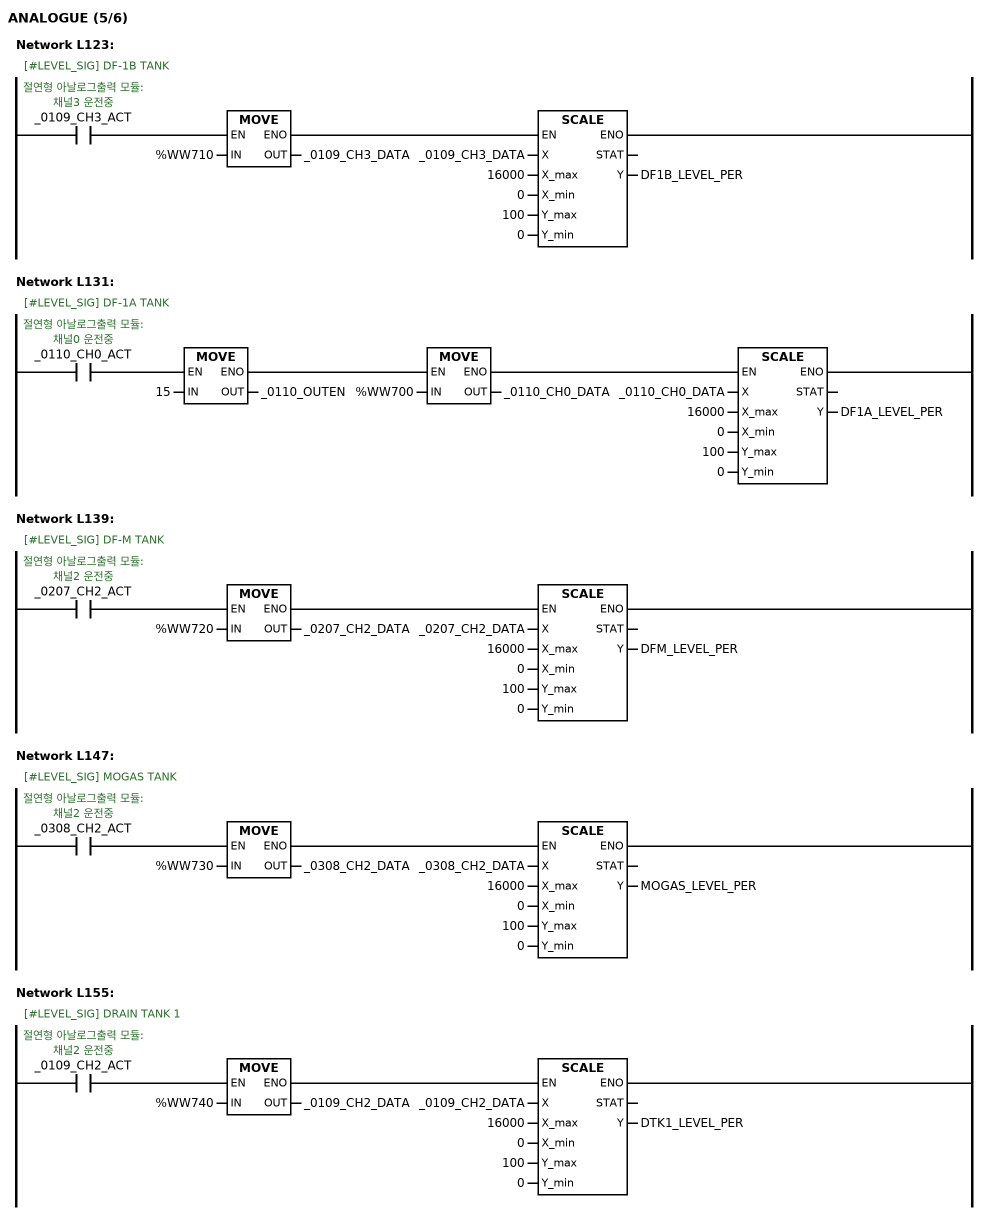
(* [#LEVEL_SIG] DF-1B TANK *)
(* Rung L123 *)
IF _0109_CH3_ACT THEN
    _0109_CH3_DATA := %WW710;
    SCALE(X := _0109_CH3_DATA, X_max := 16000, X_min := 0, Y_max := 100, Y_min := 0, Y => DF1B_LEVEL_PER);
END_IF;
(* [#LEVEL_SIG] DF-1A TANK *)
(* Rung L131 *)
IF _0110_CH0_ACT THEN
    _0110_OUTEN := 15;
    _0110_CH0_DATA := %WW700;
    SCALE(X := _0110_CH0_DATA, X_max := 16000, X_min := 0, Y_max := 100, Y_min := 0, Y => DF1A_LEVEL_PER);
END_IF;
(* [#LEVEL_SIG] DF-M TANK *)
(* Rung L139 *)
IF _0207_CH2_ACT THEN
    _0207_CH2_DATA := %WW720;
    SCALE(X := _0207_CH2_DATA, X_max := 16000, X_min := 0, Y_max := 100, Y_min := 0, Y => DFM_LEVEL_PER);
END_IF;
(* [#LEVEL_SIG] MOGAS TANK *)
(* Rung L147 *)
IF _0308_CH2_ACT THEN
    _0308_CH2_DATA := %WW730;
    SCALE(X := _0308_CH2_DATA, X_max := 16000, X_min := 0, Y_max := 100, Y_min := 0, Y => MOGAS_LEVEL_PER);
END_IF;
(* [#LEVEL_SIG] DRAIN TANK 1 *)
(* Rung L155 *)
IF _0109_CH2_ACT THEN
    _0109_CH2_DATA := %WW740;
    SCALE(X := _0109_CH2_DATA, X_max := 16000, X_min := 0, Y_max := 100, Y_min := 0, Y => DTK1_LEVEL_PER);
END_IF;

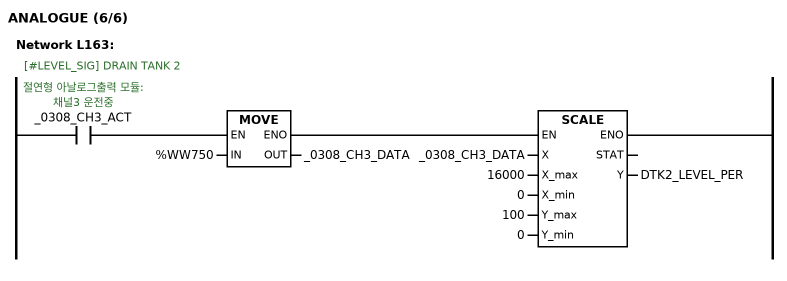
(* [#LEVEL_SIG] DRAIN TANK 2 *)
(* Rung L163 *)
IF _0308_CH3_ACT THEN
    _0308_CH3_DATA := %WW750;
    SCALE(X := _0308_CH3_DATA, X_max := 16000, X_min := 0, Y_max := 100, Y_min := 0, Y => DTK2_LEVEL_PER);
END_IF;
END_PROGRAM

PROGRAM COMMUNICATION (* task: 스캔 프로그램 *)

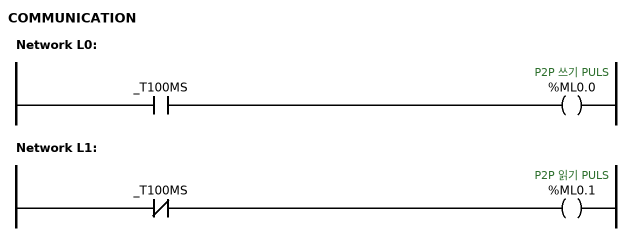
(* Rung L0 *)
%ML0.0 := _T100MS;
(* Rung L1 *)
%ML0.1 := NOT _T100MS;
END_PROGRAM

PROGRAM SCADA (* task: 스캔 프로그램 *)
VAR
    DFM_anyRun_SW : BOOL;
    MOGAS_anyRun_SW : BOOL;
END_VAR
VAR
    _t1 : BOOL;
    _t2 : BOOL;
END_VAR

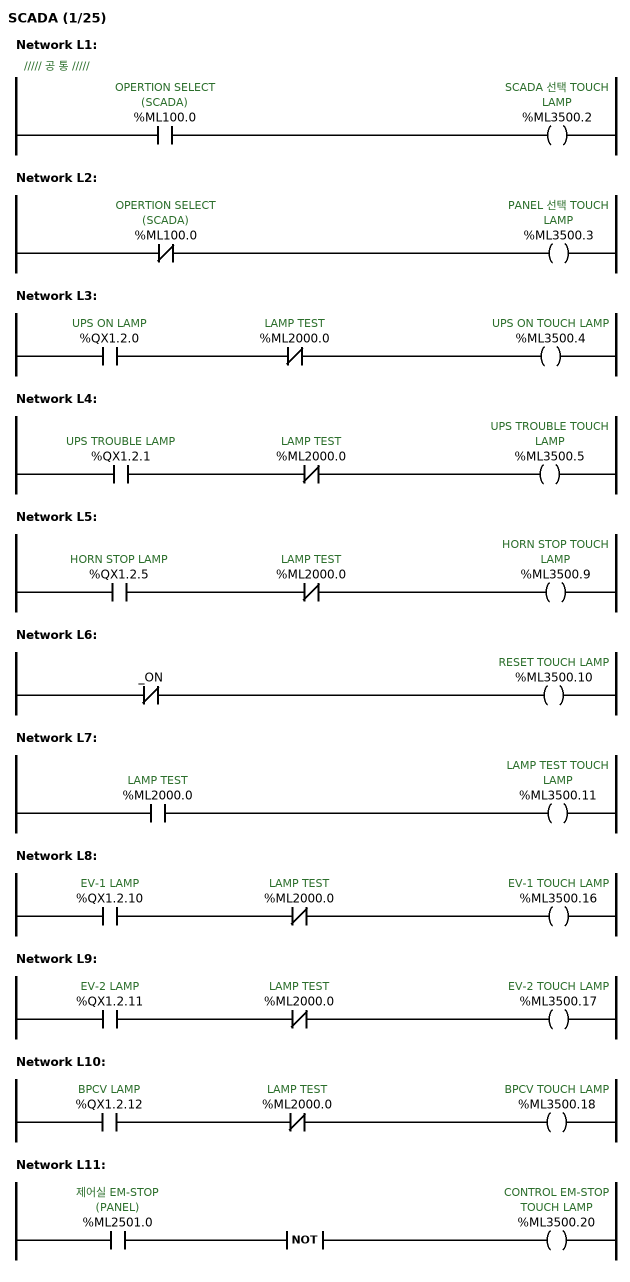
(* ///// 공 통 ///// *)
(* Rung L1 *)
%ML3500.2 := %ML100.0;
(* Rung L2 *)
%ML3500.3 := NOT %ML100.0;
(* Rung L3 *)
%ML3500.4 := %QX1.2.0 AND NOT %ML2000.0;
(* Rung L4 *)
%ML3500.5 := %QX1.2.1 AND NOT %ML2000.0;
(* Rung L5 *)
%ML3500.9 := %QX1.2.5 AND NOT %ML2000.0;
(* Rung L6 *)
%ML3500.10 := NOT _ON;
(* Rung L7 *)
%ML3500.11 := %ML2000.0;
(* Rung L8 *)
%ML3500.16 := %QX1.2.10 AND NOT %ML2000.0;
(* Rung L9 *)
%ML3500.17 := %QX1.2.11 AND NOT %ML2000.0;
(* Rung L10 *)
%ML3500.18 := %QX1.2.12 AND NOT %ML2000.0;
(* Rung L11 *)
%ML3500.20 := NOT %ML2501.0;

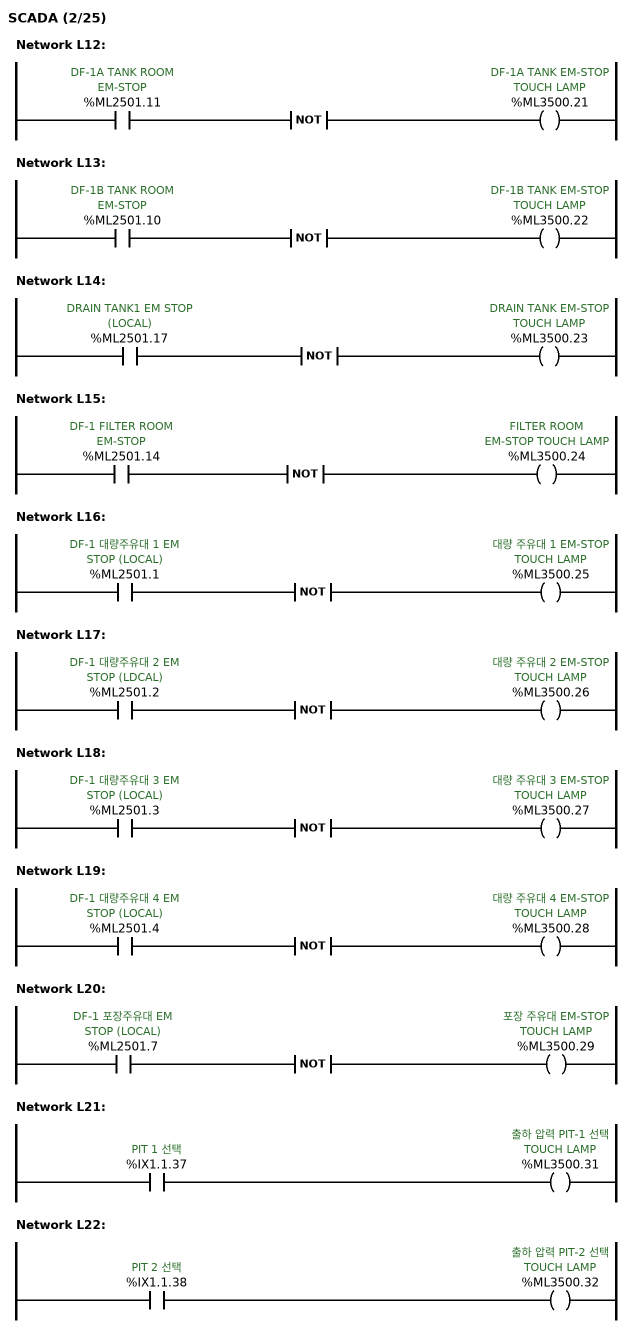
(* Rung L12 *)
%ML3500.21 := NOT %ML2501.11;
(* Rung L13 *)
%ML3500.22 := NOT %ML2501.10;
(* Rung L14 *)
%ML3500.23 := NOT %ML2501.17;
(* Rung L15 *)
%ML3500.24 := NOT %ML2501.14;
(* Rung L16 *)
%ML3500.25 := NOT %ML2501.1;
(* Rung L17 *)
%ML3500.26 := NOT %ML2501.2;
(* Rung L18 *)
%ML3500.27 := NOT %ML2501.3;
(* Rung L19 *)
%ML3500.28 := NOT %ML2501.4;
(* Rung L20 *)
%ML3500.29 := NOT %ML2501.7;
(* Rung L21 *)
%ML3500.31 := %IX1.1.37;
(* Rung L22 *)
%ML3500.32 := %IX1.1.38;

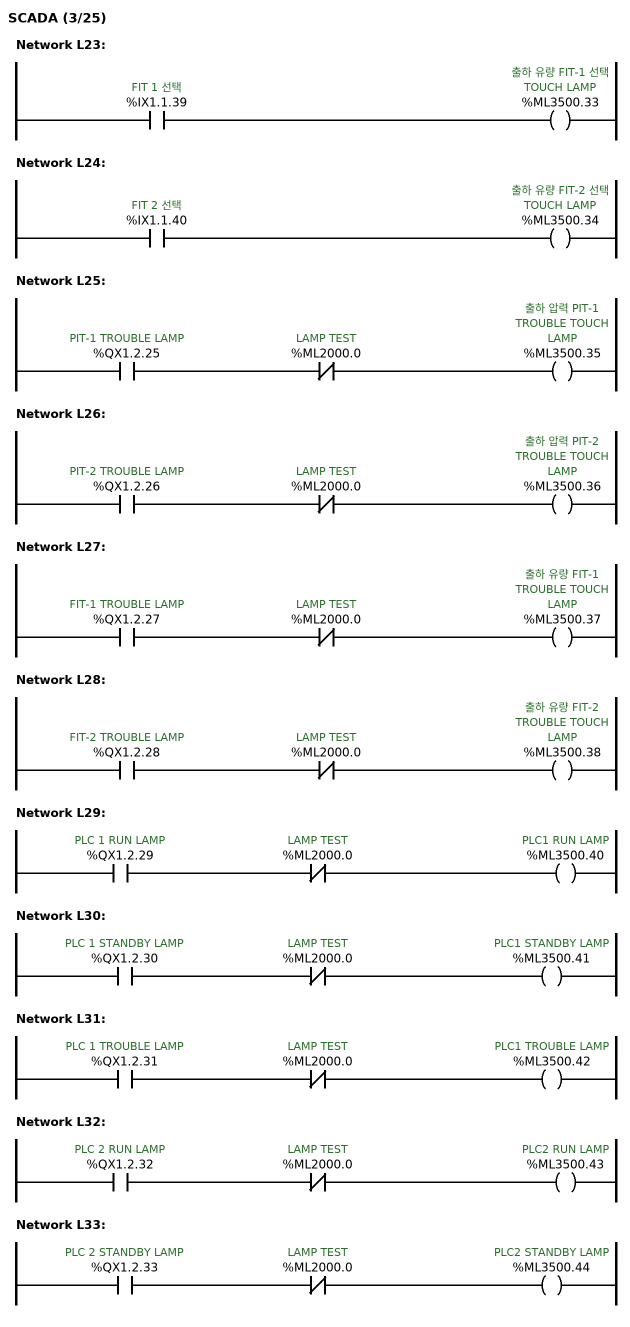
(* Rung L23 *)
%ML3500.33 := %IX1.1.39;
(* Rung L24 *)
%ML3500.34 := %IX1.1.40;
(* Rung L25 *)
%ML3500.35 := %QX1.2.25 AND NOT %ML2000.0;
(* Rung L26 *)
%ML3500.36 := %QX1.2.26 AND NOT %ML2000.0;
(* Rung L27 *)
%ML3500.37 := %QX1.2.27 AND NOT %ML2000.0;
(* Rung L28 *)
%ML3500.38 := %QX1.2.28 AND NOT %ML2000.0;
(* Rung L29 *)
%ML3500.40 := %QX1.2.29 AND NOT %ML2000.0;
(* Rung L30 *)
%ML3500.41 := %QX1.2.30 AND NOT %ML2000.0;
(* Rung L31 *)
%ML3500.42 := %QX1.2.31 AND NOT %ML2000.0;
(* Rung L32 *)
%ML3500.43 := %QX1.2.32 AND NOT %ML2000.0;
(* Rung L33 *)
%ML3500.44 := %QX1.2.33 AND NOT %ML2000.0;

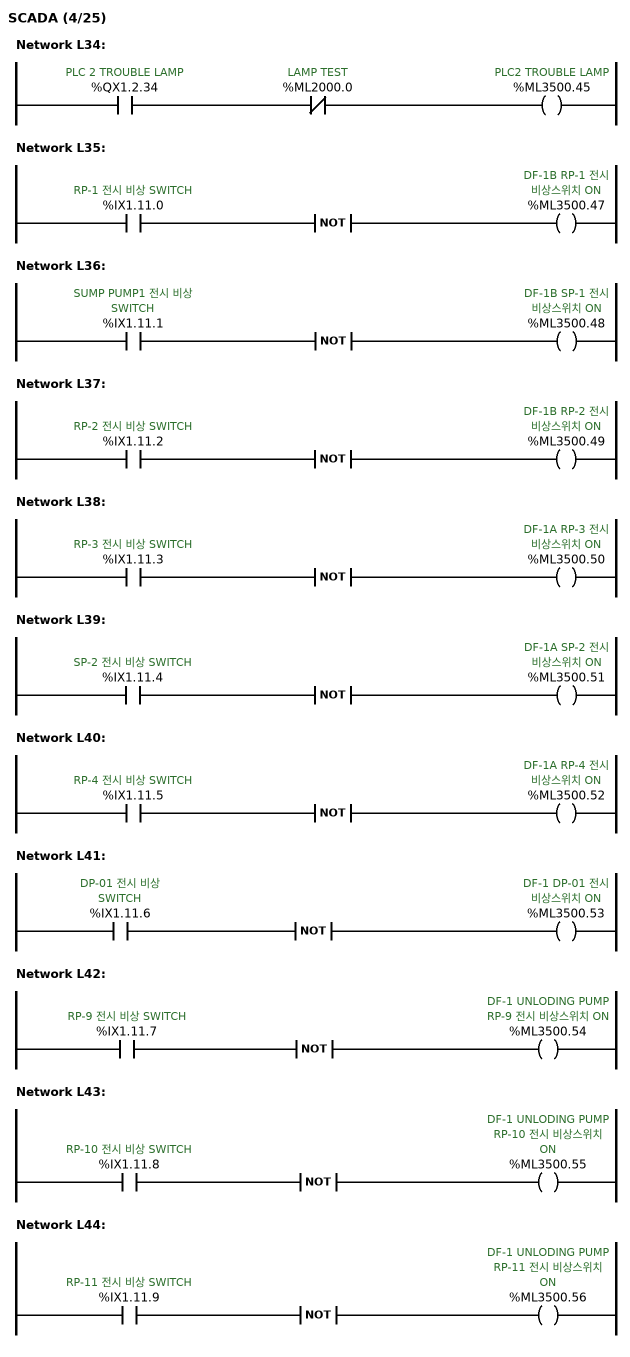
(* Rung L34 *)
%ML3500.45 := %QX1.2.34 AND NOT %ML2000.0;
(* Rung L35 *)
%ML3500.47 := NOT %IX1.11.0;
(* Rung L36 *)
%ML3500.48 := NOT %IX1.11.1;
(* Rung L37 *)
%ML3500.49 := NOT %IX1.11.2;
(* Rung L38 *)
%ML3500.50 := NOT %IX1.11.3;
(* Rung L39 *)
%ML3500.51 := NOT %IX1.11.4;
(* Rung L40 *)
%ML3500.52 := NOT %IX1.11.5;
(* Rung L41 *)
%ML3500.53 := NOT %IX1.11.6;
(* Rung L42 *)
%ML3500.54 := NOT %IX1.11.7;
(* Rung L43 *)
%ML3500.55 := NOT %IX1.11.8;
(* Rung L44 *)
%ML3500.56 := NOT %IX1.11.9;

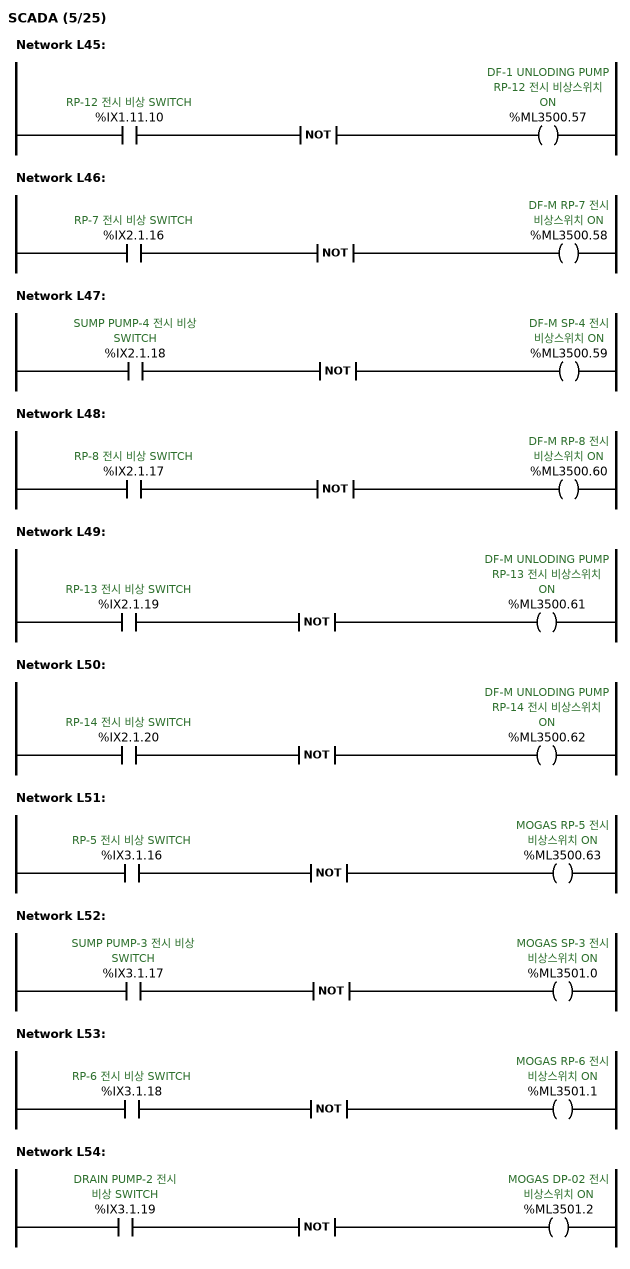
(* Rung L45 *)
%ML3500.57 := NOT %IX1.11.10;
(* Rung L46 *)
%ML3500.58 := NOT %IX2.1.16;
(* Rung L47 *)
%ML3500.59 := NOT %IX2.1.18;
(* Rung L48 *)
%ML3500.60 := NOT %IX2.1.17;
(* Rung L49 *)
%ML3500.61 := NOT %IX2.1.19;
(* Rung L50 *)
%ML3500.62 := NOT %IX2.1.20;
(* Rung L51 *)
%ML3500.63 := NOT %IX3.1.16;
(* Rung L52 *)
%ML3501.0 := NOT %IX3.1.17;
(* Rung L53 *)
%ML3501.1 := NOT %IX3.1.18;
(* Rung L54 *)
%ML3501.2 := NOT %IX3.1.19;

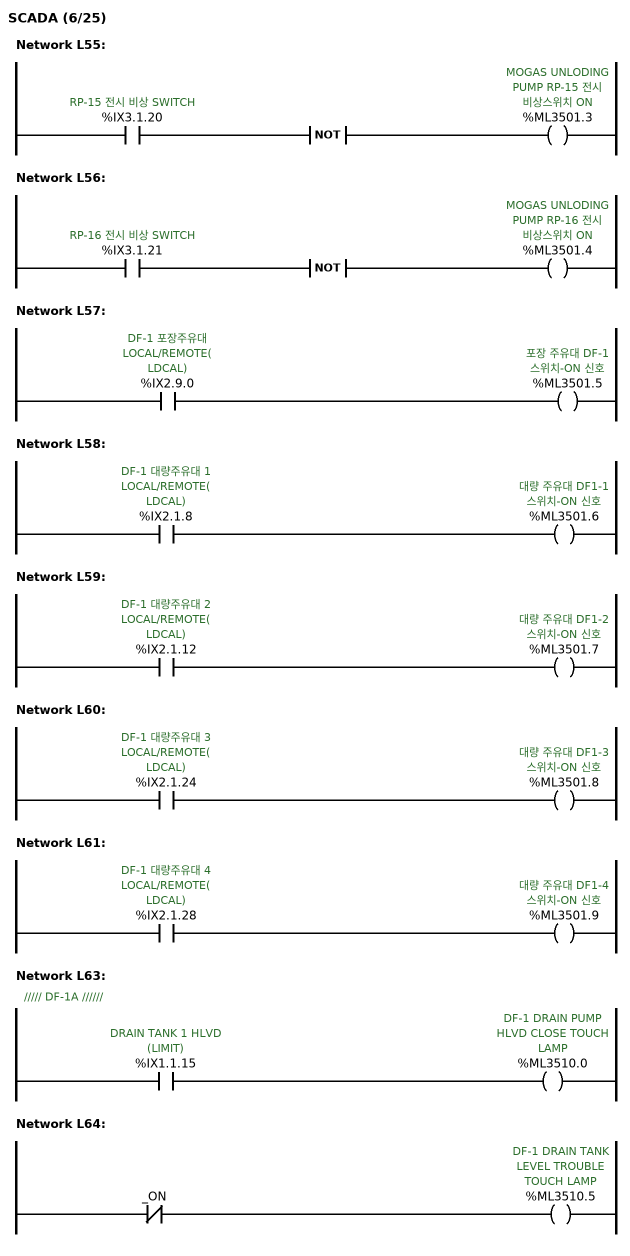
(* Rung L55 *)
%ML3501.3 := NOT %IX3.1.20;
(* Rung L56 *)
%ML3501.4 := NOT %IX3.1.21;
(* Rung L57 *)
%ML3501.5 := %IX2.9.0;
(* Rung L58 *)
%ML3501.6 := %IX2.1.8;
(* Rung L59 *)
%ML3501.7 := %IX2.1.12;
(* Rung L60 *)
%ML3501.8 := %IX2.1.24;
(* Rung L61 *)
%ML3501.9 := %IX2.1.28;
(* ///// DF-1A ////// *)
(* Rung L63 *)
%ML3510.0 := %IX1.1.15;
(* Rung L64 *)
%ML3510.5 := NOT _ON;

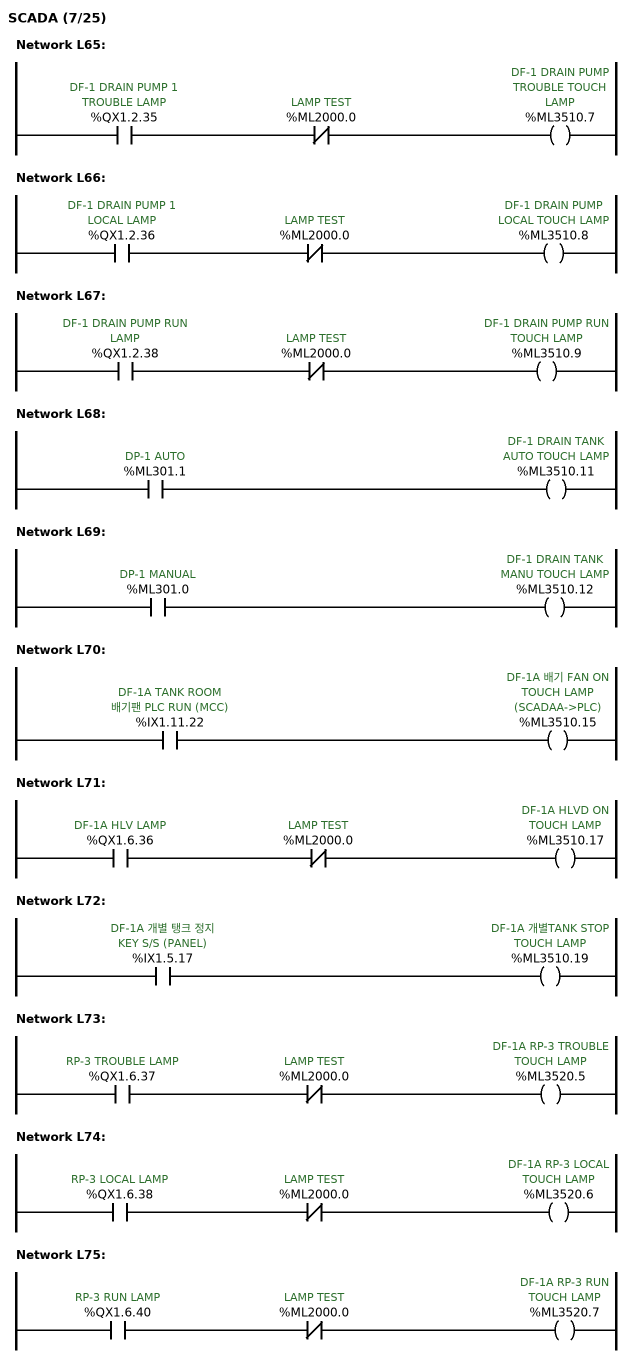
(* Rung L65 *)
%ML3510.7 := %QX1.2.35 AND NOT %ML2000.0;
(* Rung L66 *)
%ML3510.8 := %QX1.2.36 AND NOT %ML2000.0;
(* Rung L67 *)
%ML3510.9 := %QX1.2.38 AND NOT %ML2000.0;
(* Rung L68 *)
%ML3510.11 := %ML301.1;
(* Rung L69 *)
%ML3510.12 := %ML301.0;
(* Rung L70 *)
%ML3510.15 := %IX1.11.22;
(* Rung L71 *)
%ML3510.17 := %QX1.6.36 AND NOT %ML2000.0;
(* Rung L72 *)
%ML3510.19 := %IX1.5.17;
(* Rung L73 *)
%ML3520.5 := %QX1.6.37 AND NOT %ML2000.0;
(* Rung L74 *)
%ML3520.6 := %QX1.6.38 AND NOT %ML2000.0;
(* Rung L75 *)
%ML3520.7 := %QX1.6.40 AND NOT %ML2000.0;

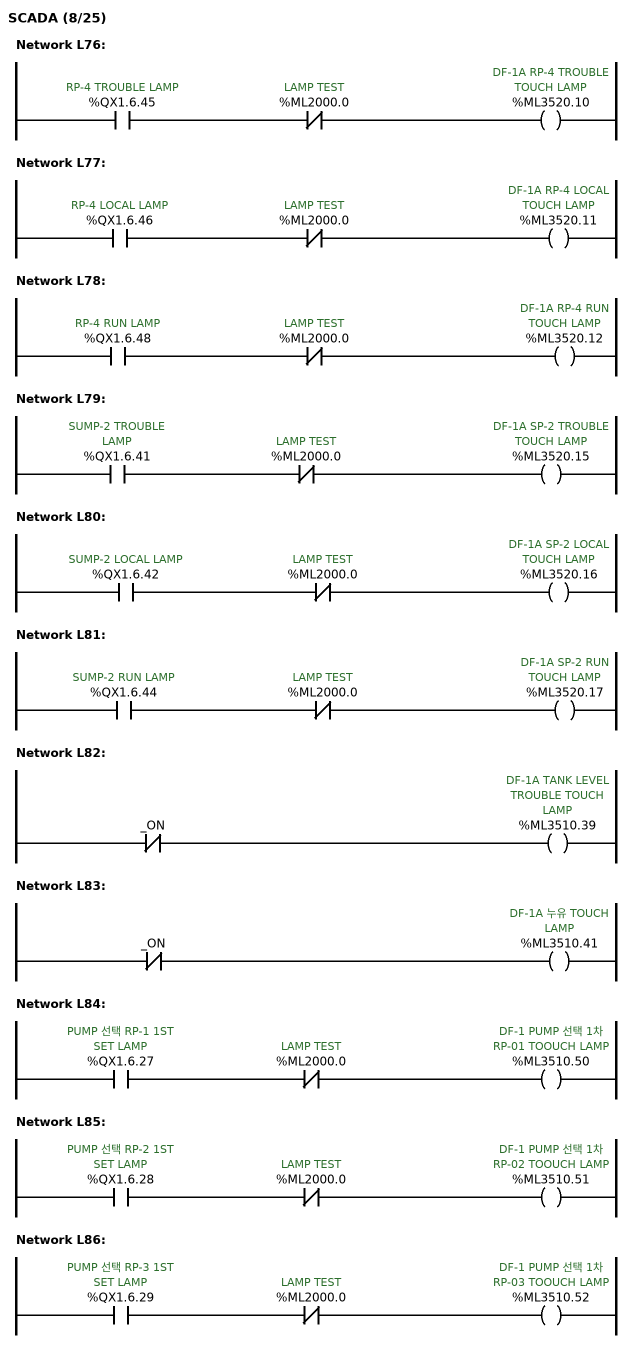
(* Rung L76 *)
%ML3520.10 := %QX1.6.45 AND NOT %ML2000.0;
(* Rung L77 *)
%ML3520.11 := %QX1.6.46 AND NOT %ML2000.0;
(* Rung L78 *)
%ML3520.12 := %QX1.6.48 AND NOT %ML2000.0;
(* Rung L79 *)
%ML3520.15 := %QX1.6.41 AND NOT %ML2000.0;
(* Rung L80 *)
%ML3520.16 := %QX1.6.42 AND NOT %ML2000.0;
(* Rung L81 *)
%ML3520.17 := %QX1.6.44 AND NOT %ML2000.0;
(* Rung L82 *)
%ML3510.39 := NOT _ON;
(* Rung L83 *)
%ML3510.41 := NOT _ON;
(* Rung L84 *)
%ML3510.50 := %QX1.6.27 AND NOT %ML2000.0;
(* Rung L85 *)
%ML3510.51 := %QX1.6.28 AND NOT %ML2000.0;
(* Rung L86 *)
%ML3510.52 := %QX1.6.29 AND NOT %ML2000.0;

